SPLINE
SPL {X  -156.487, Y  +349.204, Z    +0.000, E1   -21.338, E3 -341381.497}
SPL {X  -159.136, Y  +365.992, Z    +0.000, E1   -12.463, E3 -341392.255}
SPL {X  -159.799, Y  +374.694, Z    +0.000, E1    -7.504, E3 -341395.359}
SPL {X  -159.976, Y  +380.404, Z    +0.000, E1    -3.959, E3 -341396.892}
SPL {X  -159.990, Y  +384.773, Z    +0.000, E1    -1.003, E3 -341397.786}
SPL {X  -159.990, Y  +387.968, Z    +0.000, E1    +1.448, E3 -341398.355}
SPL {X  -159.990, Y  +391.397, Z    +0.000, E1    +4.422, E3 -341398.979}
SPL {X  -159.990, Y  +395.864, Z    +0.000, E1    +8.712, E3 -341400.067}
SPL {X  -159.990, Y  +401.273, Z    +0.000, E1   +14.176, E3 -341401.795}
SPL {X  -159.990, Y  +411.788, Z    +0.000, E1   +23.693, E3 -341407.338}
SPL {X  -159.990, Y  +438.158, Z    +0.000, E1   +37.630, E3 -341430.615}
SPL {X  -159.990, Y  +468.567, Z    +0.000, E1   +41.922, E3 -341479.959}
SPL {X  -159.990, Y  +474.616, Z    +0.000, E1   +41.909, E3 -341494.288}
SPL {X  -159.990, Y  +481.610, Z    +0.000, E1   +41.947, E3 -341510.775}
SPL {X  -159.990, Y  +488.618, Z    +0.000, E1   +41.913, E3 -341527.387}
SPL {X  -159.990, Y  +494.299, Z    +0.000, E1   +41.910, E3 -341540.821}
SPL {X  -159.990, Y  +499.538, Z    +0.000, E1   +41.904, E3 -341553.216}
SPL {X  -159.990, Y  +505.259, Z    +0.000, E1   +41.922, E3 -341566.715}
SPL {X  -159.990, Y  +511.862, Z    +0.000, E1   +41.927, E3 -341582.325}
SPL {X  -159.990, Y  +517.450, Z    +0.000, E1   +41.901, E3 -341595.573}
SPL {X  -159.990, Y  +523.027, Z    +0.000, E1   +41.926, E3 -341608.717}
SPL {X  -159.990, Y  +528.611, Z    +0.000, E1   +41.900, E3 -341621.972}
SPL {X  -159.990, Y  +533.758, Z    +0.000, E1   +41.910, E3 -341634.121}
SPL {X  -159.990, Y  +539.474, Z    +0.000, E1   +41.912, E3 -341647.649}
SPL {X  -159.990, Y  +544.879, Z    +0.000, E1   +41.899, E3 -341660.460}
SPL {X  -159.990, Y  +550.802, Z    +0.000, E1   +41.920, E3 -341674.442}
SPL {X  -159.990, Y  +556.952, Z    +0.000, E1   +41.911, E3 -341688.981}
SPL {X  -159.990, Y  +562.629, Z    +0.000, E1   +41.910, E3 -341702.399}
SPL {X  -159.990, Y  +567.682, Z    +0.000, E1   +41.901, E3 -341714.358}
SPL {X  -159.990, Y  +572.912, Z    +0.000, E1   +41.914, E3 -341726.705}
SPL {X  -159.990, Y  +578.863, Z    +0.000, E1   +41.918, E3 -341740.769}
SPL {X  -159.990, Y  +584.320, Z    +0.000, E1   +41.901, E3 -341753.716}
SPL {X  -159.990, Y  +589.217, Z    +0.000, E1   +41.901, E3 -341765.289}
SPL {X  -159.990, Y  +594.252, Z    +0.000, E1   +41.903, E3 -341777.203}
SPL {X  -159.990, Y  +598.793, Z    +0.000, E1   +41.896, E3 -341787.957}
SPL {X  -159.990, Y  +604.215, Z    +0.000, E1   +41.919, E3 -341800.737}
SPL {X  -159.990, Y  +610.545, Z    +0.000, E1   +41.917, E3 -341815.707}
SPL {X  -159.990, Y  +615.720, Z    +0.000, E1   +41.899, E3 -341827.967}
SPL {X  -159.990, Y  +620.005, Z    +0.000, E1   +41.900, E3 -341838.100}
SPL {X  -159.990, Y  +624.919, Z    +0.000, E1   +41.912, E3 -341849.707}
SPL {X  -159.990, Y  +630.816, Z    +0.000, E1   +41.915, E3 -341863.636}
SPL {X  -159.990, Y  +637.009, Z    +0.000, E1   +41.925, E3 -341878.262}
SPL {X  -159.990, Y  +642.624, Z    +0.000, E1   +41.901, E3 -341891.583}
SPL {X  -159.990, Y  +647.782, Z    +0.000, E1   +41.914, E3 -341903.751}
SPL {X  -159.990, Y  +653.094, Z    +0.000, E1   +41.905, E3 -341916.329}
SPL {X  -159.990, Y  +657.893, Z    +0.000, E1   +41.899, E3 -341927.695}
SPL {X  -159.990, Y  +662.516, Z    +0.000, E1   +41.899, E3 -341938.626}
SPL {X  -159.990, Y  +668.411, Z    +0.000, E1   +41.929, E3 -341952.520}
SPL {X  -159.968, Y  +674.139, Z    +0.000, E1   +41.898, E3 -341966.124}
SPL {X  -159.817, Y  +678.937, Z    +0.000, E1   +41.879, E3 -341977.620}
SPL {X  -159.484, Y  +684.213, Z    +0.000, E1   +41.818, E3 -341990.456}
SPL {X  -159.007, Y  +689.209, Z    +0.000, E1   +41.732, E3 -342002.761}
SPL {X  -158.327, Y  +694.511, Z    +0.000, E1   +41.622, E3 -342016.012}
SPL {X  -157.480, Y  +699.729, Z    +0.000, E1   +41.453, E3 -342029.275}
SPL {X  -156.604, Y  +704.242, Z    +0.000, E1   +41.288, E3 -342040.884}
SPL {X  -155.514, Y  +709.078, Z    +0.000, E1   +41.107, E3 -342053.437}
SPL {X  -154.232, Y  +714.035, Z    +0.000, E1   +40.861, E3 -342066.496}
SPL {X  -153.147, Y  +717.790, Z    +0.000, E1   +40.640, E3 -342076.515}
SPL {X  -151.881, Y  +721.788, Z    +0.000, E1   +40.435, E3 -342087.201}
SPL {X  -148.572, Y  +730.857, Z    +0.000, E1   +36.304, E3 -342143.410}
ENDSPLINE

SPLINE
SPL {X  -156.377, Y  +705.307, Z    +0.000, E1   +21.740, E3 -342197.659}
SPL {X  -159.301, Y  +686.331, Z    +0.000, E1   +11.648, E3 -342210.303}
SPL {X  -159.936, Y  +675.651, Z    +0.000, E1    +5.377, E3 -342214.019}
SPL {X  -159.990, Y  +670.142, Z    +0.000, E1    +1.740, E3 -342215.318}
SPL {X  -159.990, Y  +666.629, Z    +0.000, E1    -0.827, E3 -342215.968}
SPL {X  -159.990, Y  +662.407, Z    +0.000, E1    -4.406, E3 -342216.818}
SPL {X  -159.990, Y  +657.382, Z    +0.000, E1    -9.217, E3 -342218.200}
SPL {X  -159.990, Y  +653.255, Z    +0.000, E1   -13.347, E3 -342219.529}
SPL {X  -159.990, Y  +646.242, Z    +0.000, E1   -19.956, E3 -342222.603}
SPL {X  -159.990, Y  +624.365, Z    +0.000, E1   -33.860, E3 -342240.504}
SPL {X  -159.990, Y  +615.596, Z    +0.000, E1   -36.980, E3 -342250.163}
SPL {X  -159.990, Y  +586.905, Z    +0.000, E1   -41.264, E3 -342297.189}
SPL {X  -159.990, Y  +581.111, Z    +0.000, E1   -41.245, E3 -342311.243}
SPL {X  -159.990, Y  +576.269, Z    +0.000, E1   -41.239, E3 -342322.971}
SPL {X  -159.990, Y  +571.714, Z    +0.000, E1   -41.240, E3 -342333.999}
SPL {X  -159.990, Y  +567.050, Z    +0.000, E1   -41.238, E3 -342345.286}
SPL {X  -159.990, Y  +561.959, Z    +0.000, E1   -41.251, E3 -342357.584}
SPL {X  -159.990, Y  +557.719, Z    +0.000, E1   -41.226, E3 -342367.886}
SPL {X  -159.990, Y  +554.148, Z    +0.000, E1   -41.237, E3 -342376.502}
SPL {X  -159.990, Y  +548.812, Z    +0.000, E1   -41.263, E3 -342389.376}
SPL {X  -159.990, Y  +543.804, Z    +0.000, E1   -41.237, E3 -342401.541}
SPL {X  -159.990, Y  +538.952, Z    +0.000, E1   -41.247, E3 -342413.288}
SPL {X  -159.990, Y  +534.225, Z    +0.000, E1   -41.236, E3 -342424.721}
SPL {X  -159.990, Y  +529.136, Z    +0.000, E1   -41.262, E3 -342436.997}
SPL {X  -159.990, Y  +522.690, Z    +0.000, E1   -41.265, E3 -342452.597}
SPL {X  -159.990, Y  +516.698, Z    +0.000, E1   -41.259, E3 -342467.071}
SPL {X  -159.990, Y  +510.896, Z    +0.000, E1   -41.267, E3 -342481.089}
SPL {X  -159.990, Y  +505.215, Z    +0.000, E1   -41.261, E3 -342494.849}
SPL {X  -159.990, Y  +500.102, Z    +0.000, E1   -41.251, E3 -342507.232}
SPL {X  -159.990, Y  +495.023, Z    +0.000, E1   -41.263, E3 -342519.481}
SPL {X  -159.990, Y  +479.011, Z    +0.000, E1   -45.740, E3 -342528.863}
SPL {X  -159.990, Y  +471.379, Z    +0.000, E1   -46.435, E3 -342540.479}
SPL {X  -159.990, Y  +465.881, Z    +0.000, E1   -45.385, E3 -342558.081}
SPL {X  -159.990, Y  +461.571, Z    +0.000, E1   -44.440, E3 -342572.607}
SPL {X  -159.990, Y  +458.229, Z    +0.000, E1   -43.579, E3 -342585.141}
SPL {X  -159.990, Y  +453.434, Z    +0.000, E1   -43.227, E3 -342597.915}
SPL {X  -159.990, Y  +448.702, Z    +0.000, E1   -43.218, E3 -342608.637}
SPL {X  -159.990, Y  +442.224, Z    +0.000, E1   -43.270, E3 -342623.187}
SPL {X  -159.990, Y  +435.724, Z    +0.000, E1   -43.218, E3 -342637.945}
SPL {X  -159.990, Y  +430.527, Z    +0.000, E1   -43.236, E3 -342649.634}
SPL {X  -159.990, Y  +424.433, Z    +0.000, E1   -43.237, E3 -342663.383}
SPL {X  -159.990, Y  +419.466, Z    +0.000, E1   -43.217, E3 -342674.623}
SPL {X  -159.990, Y  +414.585, Z    +0.000, E1   -43.233, E3 -342685.615}
SPL {X  -159.990, Y  +409.927, Z    +0.000, E1   -43.217, E3 -342696.147}
SPL {X  -159.990, Y  +405.428, Z    +0.000, E1   -43.230, E3 -342706.305}
SPL {X  -159.990, Y  +398.518, Z    +0.000, E1   -43.261, E3 -342721.859}
SPL {X  -159.990, Y  +392.163, Z    +0.000, E1   -43.223, E3 -342736.259}
SPL {X  -159.990, Y  +387.342, Z    +0.000, E1   -43.224, E3 -342747.137}
SPL {X  -159.990, Y  +382.548, Z    +0.000, E1   -43.224, E3 -342757.959}
SPL {X  -159.922, Y  +377.835, Z    +0.000, E1   -43.211, E3 -342768.676}
SPL {X  -159.712, Y  +373.072, Z    +0.000, E1   -43.177, E3 -342779.642}
SPL {X  -159.289, Y  +367.537, Z    +0.000, E1   -43.118, E3 -342792.554}
SPL {X  -158.730, Y  +362.464, Z    +0.000, E1   -43.003, E3 -342804.586}
SPL {X  -158.182, Y  +358.518, Z    +0.000, E1   -42.902, E3 -342814.064}
SPL {X  -157.507, Y  +354.423, Z    +0.000, E1   -42.786, E3 -342824.010}
SPL {X  -156.676, Y  +350.104, Z    +0.000, E1   -42.637, E3 -342834.615}
SPL {X  -155.489, Y  +344.819, Z    +0.000, E1   -42.446, E3 -342847.738}
SPL {X  -153.911, Y  +338.816, Z    +0.000, E1   -42.155, E3 -342862.914}
SPL {X  -152.412, Y  +333.846, Z    +0.000, E1   -41.856, E3 -342875.685}
SPL {X  -151.009, Y  +329.651, Z    +0.000, E1   -41.581, E3 -342886.585}
SPL {X  -148.356, Y  +322.607, Z    +0.000, E1   -36.121, E3 -342947.061}
ENDSPLINE

SPLINE
SPL {X  -156.487, Y  +349.204, Z    +0.000, E1   -21.338, E3 -343002.186}
SPL {X  -159.136, Y  +365.992, Z    +0.000, E1   -12.463, E3 -343012.945}
SPL {X  -159.799, Y  +374.694, Z    +0.000, E1    -7.504, E3 -343016.049}
SPL {X  -159.976, Y  +380.404, Z    +0.000, E1    -3.959, E3 -343017.582}
SPL {X  -159.990, Y  +384.773, Z    +0.000, E1    -1.003, E3 -343018.476}
SPL {X  -159.990, Y  +387.968, Z    +0.000, E1    +1.448, E3 -343019.044}
SPL {X  -159.990, Y  +391.397, Z    +0.000, E1    +4.422, E3 -343019.668}
SPL {X  -159.990, Y  +395.864, Z    +0.000, E1    +8.712, E3 -343020.757}
SPL {X  -159.990, Y  +401.273, Z    +0.000, E1   +14.176, E3 -343022.484}
SPL {X  -159.990, Y  +411.788, Z    +0.000, E1   +23.693, E3 -343028.027}
SPL {X  -159.990, Y  +438.158, Z    +0.000, E1   +37.630, E3 -343051.304}
SPL {X  -159.990, Y  +468.567, Z    +0.000, E1   +41.922, E3 -343100.648}
SPL {X  -159.990, Y  +474.616, Z    +0.000, E1   +41.909, E3 -343114.978}
SPL {X  -159.990, Y  +478.952, Z    +0.000, E1   +41.885, E3 -343125.276}
SPL {X  -159.990, Y  +484.724, Z    +0.000, E1   +41.943, E3 -343138.827}
SPL {X  -159.990, Y  +492.944, Z    +0.000, E1   +41.952, E3 -343158.247}
SPL {X  -159.990, Y  +499.538, Z    +0.000, E1   +41.904, E3 -343173.905}
SPL {X  -159.990, Y  +505.259, Z    +0.000, E1   +41.922, E3 -343187.405}
SPL {X  -159.990, Y  +511.862, Z    +0.000, E1   +41.927, E3 -343203.015}
SPL {X  -159.990, Y  +517.450, Z    +0.000, E1   +41.901, E3 -343216.262}
SPL {X  -159.990, Y  +523.027, Z    +0.000, E1   +41.926, E3 -343229.407}
SPL {X  -159.990, Y  +528.611, Z    +0.000, E1   +41.900, E3 -343242.662}
SPL {X  -159.990, Y  +533.758, Z    +0.000, E1   +41.910, E3 -343254.811}
SPL {X  -159.990, Y  +539.474, Z    +0.000, E1   +41.912, E3 -343268.338}
SPL {X  -159.990, Y  +544.879, Z    +0.000, E1   +41.899, E3 -343281.150}
SPL {X  -159.990, Y  +550.802, Z    +0.000, E1   +41.920, E3 -343295.131}
SPL {X  -159.990, Y  +556.952, Z    +0.000, E1   +41.911, E3 -343309.670}
SPL {X  -159.990, Y  +562.629, Z    +0.000, E1   +41.910, E3 -343323.088}
SPL {X  -159.990, Y  +569.054, Z    +0.000, E1   +41.933, E3 -343338.243}
SPL {X  -159.990, Y  +575.562, Z    +0.000, E1   +41.916, E3 -343353.656}
SPL {X  -159.990, Y  +580.118, Z    +0.000, E1   +41.891, E3 -343364.469}
SPL {X  -159.990, Y  +584.320, Z    +0.000, E1   +41.901, E3 -343374.405}
SPL {X  -159.990, Y  +589.217, Z    +0.000, E1   +41.901, E3 -343385.978}
SPL {X  -159.990, Y  +594.252, Z    +0.000, E1   +41.903, E3 -343397.893}
SPL {X  -159.990, Y  +598.793, Z    +0.000, E1   +41.896, E3 -343408.647}
SPL {X  -159.990, Y  +604.215, Z    +0.000, E1   +41.919, E3 -343421.427}
SPL {X  -159.990, Y  +609.216, Z    +0.000, E1   +41.890, E3 -343433.295}
SPL {X  -159.990, Y  +614.570, Z    +0.000, E1   +41.926, E3 -343445.900}
SPL {X  -159.990, Y  +620.005, Z    +0.000, E1   +41.900, E3 -343458.790}
SPL {X  -159.990, Y  +624.919, Z    +0.000, E1   +41.912, E3 -343470.397}
SPL {X  -159.990, Y  +630.816, Z    +0.000, E1   +41.915, E3 -343484.326}
SPL {X  -159.990, Y  +635.747, Z    +0.000, E1   +41.898, E3 -343496.005}
SPL {X  -159.990, Y  +641.479, Z    +0.000, E1   +41.931, E3 -343509.519}
SPL {X  -159.990, Y  +647.782, Z    +0.000, E1   +41.914, E3 -343524.441}
SPL {X  -159.990, Y  +653.094, Z    +0.000, E1   +41.905, E3 -343537.019}
SPL {X  -159.990, Y  +657.893, Z    +0.000, E1   +41.899, E3 -343548.385}
SPL {X  -159.990, Y  +662.516, Z    +0.000, E1   +41.899, E3 -343559.316}
SPL {X  -159.990, Y  +668.411, Z    +0.000, E1   +41.929, E3 -343573.210}
SPL {X  -159.968, Y  +674.139, Z    +0.000, E1   +41.898, E3 -343586.814}
SPL {X  -159.817, Y  +678.937, Z    +0.000, E1   +41.879, E3 -343598.310}
SPL {X  -159.484, Y  +684.213, Z    +0.000, E1   +41.818, E3 -343611.146}
SPL {X  -159.007, Y  +689.209, Z    +0.000, E1   +41.732, E3 -343623.451}
SPL {X  -158.327, Y  +694.511, Z    +0.000, E1   +41.622, E3 -343636.702}
SPL {X  -157.480, Y  +699.729, Z    +0.000, E1   +41.453, E3 -343649.965}
SPL {X  -156.604, Y  +704.242, Z    +0.000, E1   +41.288, E3 -343661.573}
SPL {X  -155.514, Y  +709.078, Z    +0.000, E1   +41.107, E3 -343674.127}
SPL {X  -154.232, Y  +714.035, Z    +0.000, E1   +40.861, E3 -343687.186}
SPL {X  -153.147, Y  +717.790, Z    +0.000, E1   +40.640, E3 -343697.204}
SPL {X  -151.881, Y  +721.788, Z    +0.000, E1   +40.435, E3 -343707.891}
SPL {X  -148.572, Y  +730.857, Z    +0.000, E1   +36.304, E3 -343764.100}
ENDSPLINE

SPLINE
SPL {X  -156.377, Y  +705.307, Z    +0.000, E1   +21.740, E3 -343818.348}
SPL {X  -158.965, Y  +689.585, Z    +0.000, E1   +13.405, E3 -343829.506}
SPL {X  -159.884, Y  +677.314, Z    +0.000, E1    +6.475, E3 -343834.219}
SPL {X  -159.990, Y  +670.142, Z    +0.000, E1    +1.740, E3 -343836.008}
SPL {X  -159.990, Y  +666.629, Z    +0.000, E1    -0.827, E3 -343836.658}
SPL {X  -159.990, Y  +662.407, Z    +0.000, E1    -4.406, E3 -343837.508}
SPL {X  -159.990, Y  +657.382, Z    +0.000, E1    -9.217, E3 -343838.890}
SPL {X  -159.990, Y  +653.255, Z    +0.000, E1   -13.347, E3 -343840.219}
SPL {X  -159.990, Y  +646.242, Z    +0.000, E1   -19.956, E3 -343843.293}
SPL {X  -159.990, Y  +624.365, Z    +0.000, E1   -33.860, E3 -343861.194}
SPL {X  -159.990, Y  +615.596, Z    +0.000, E1   -36.980, E3 -343870.853}
SPL {X  -159.990, Y  +586.905, Z    +0.000, E1   -41.264, E3 -343917.879}
SPL {X  -159.990, Y  +581.111, Z    +0.000, E1   -41.245, E3 -343931.933}
SPL {X  -159.990, Y  +576.269, Z    +0.000, E1   -41.239, E3 -343943.661}
SPL {X  -159.990, Y  +571.714, Z    +0.000, E1   -41.240, E3 -343954.689}
SPL {X  -159.990, Y  +567.050, Z    +0.000, E1   -41.238, E3 -343965.975}
SPL {X  -159.990, Y  +561.959, Z    +0.000, E1   -41.251, E3 -343978.274}
SPL {X  -159.990, Y  +555.553, Z    +0.000, E1   -41.273, E3 -343993.742}
SPL {X  -159.990, Y  +549.897, Z    +0.000, E1   -41.240, E3 -344007.472}
SPL {X  -159.990, Y  +544.775, Z    +0.000, E1   -41.260, E3 -344019.847}
SPL {X  -159.990, Y  +540.176, Z    +0.000, E1   -41.224, E3 -344031.056}
SPL {X  -159.990, Y  +535.325, Z    +0.000, E1   -41.260, E3 -344042.719}
SPL {X  -159.990, Y  +529.136, Z    +0.000, E1   -41.262, E3 -344057.687}
SPL {X  -159.990, Y  +522.690, Z    +0.000, E1   -41.265, E3 -344073.287}
SPL {X  -159.990, Y  +516.698, Z    +0.000, E1   -41.259, E3 -344087.761}
SPL {X  -159.990, Y  +510.896, Z    +0.000, E1   -41.267, E3 -344101.779}
SPL {X  -159.990, Y  +505.215, Z    +0.000, E1   -41.261, E3 -344115.539}
SPL {X  -159.990, Y  +500.102, Z    +0.000, E1   -41.251, E3 -344127.922}
SPL {X  -159.990, Y  +495.023, Z    +0.000, E1   -41.263, E3 -344140.171}
SPL {X  -159.990, Y  +479.011, Z    +0.000, E1   -45.740, E3 -344149.553}
SPL {X  -159.990, Y  +471.379, Z    +0.000, E1   -46.435, E3 -344161.168}
SPL {X  -159.990, Y  +466.895, Z    +0.000, E1   -45.533, E3 -344175.573}
SPL {X  -159.990, Y  +462.409, Z    +0.000, E1   -44.664, E3 -344190.348}
SPL {X  -159.990, Y  +458.229, Z    +0.000, E1   -43.579, E3 -344205.830}
SPL {X  -159.990, Y  +453.434, Z    +0.000, E1   -43.227, E3 -344218.605}
SPL {X  -159.990, Y  +448.702, Z    +0.000, E1   -43.218, E3 -344229.326}
SPL {X  -159.990, Y  +442.224, Z    +0.000, E1   -43.270, E3 -344243.876}
SPL {X  -159.990, Y  +435.724, Z    +0.000, E1   -43.218, E3 -344258.634}
SPL {X  -159.990, Y  +430.527, Z    +0.000, E1   -43.236, E3 -344270.324}
SPL {X  -159.990, Y  +424.433, Z    +0.000, E1   -43.237, E3 -344284.073}
SPL {X  -159.990, Y  +419.466, Z    +0.000, E1   -43.217, E3 -344295.313}
SPL {X  -159.990, Y  +414.585, Z    +0.000, E1   -43.233, E3 -344306.305}
SPL {X  -159.990, Y  +409.927, Z    +0.000, E1   -43.217, E3 -344316.836}
SPL {X  -159.990, Y  +405.428, Z    +0.000, E1   -43.230, E3 -344326.994}
SPL {X  -159.990, Y  +398.518, Z    +0.000, E1   -43.261, E3 -344342.549}
SPL {X  -159.990, Y  +392.163, Z    +0.000, E1   -43.223, E3 -344356.949}
SPL {X  -159.990, Y  +387.342, Z    +0.000, E1   -43.224, E3 -344367.826}
SPL {X  -159.990, Y  +382.548, Z    +0.000, E1   -43.224, E3 -344378.649}
SPL {X  -159.922, Y  +377.835, Z    +0.000, E1   -43.211, E3 -344389.366}
SPL {X  -159.712, Y  +373.072, Z    +0.000, E1   -43.177, E3 -344400.332}
SPL {X  -159.289, Y  +367.537, Z    +0.000, E1   -43.118, E3 -344413.243}
SPL {X  -158.730, Y  +362.464, Z    +0.000, E1   -43.003, E3 -344425.275}
SPL {X  -158.182, Y  +358.518, Z    +0.000, E1   -42.902, E3 -344434.754}
SPL {X  -157.507, Y  +354.423, Z    +0.000, E1   -42.786, E3 -344444.699}
SPL {X  -156.676, Y  +350.104, Z    +0.000, E1   -42.637, E3 -344455.305}
SPL {X  -155.489, Y  +344.819, Z    +0.000, E1   -42.446, E3 -344468.428}
SPL {X  -153.911, Y  +338.816, Z    +0.000, E1   -42.155, E3 -344483.604}
SPL {X  -152.412, Y  +333.846, Z    +0.000, E1   -41.856, E3 -344496.375}
SPL {X  -151.009, Y  +329.651, Z    +0.000, E1   -41.581, E3 -344507.275}
SPL {X  -148.356, Y  +322.607, Z    +0.000, E1   -36.121, E3 -344567.750}
ENDSPLINE

SPLINE
SPL {X  -156.487, Y  +349.204, Z    +0.000, E1   -21.338, E3 -344622.876}
SPL {X  -159.136, Y  +365.992, Z    +0.000, E1   -12.463, E3 -344633.635}
SPL {X  -159.799, Y  +374.694, Z    +0.000, E1    -7.504, E3 -344636.738}
SPL {X  -159.976, Y  +380.404, Z    +0.000, E1    -3.959, E3 -344638.271}
SPL {X  -159.990, Y  +384.773, Z    +0.000, E1    -1.003, E3 -344639.166}
SPL {X  -159.990, Y  +387.968, Z    +0.000, E1    +1.448, E3 -344639.734}
SPL {X  -159.990, Y  +391.397, Z    +0.000, E1    +4.422, E3 -344640.358}
SPL {X  -159.990, Y  +395.864, Z    +0.000, E1    +8.712, E3 -344641.446}
SPL {X  -159.990, Y  +401.273, Z    +0.000, E1   +14.176, E3 -344643.174}
SPL {X  -159.990, Y  +409.369, Z    +0.000, E1   +21.807, E3 -344646.966}
SPL {X  -159.990, Y  +436.107, Z    +0.000, E1   +36.921, E3 -344669.891}
SPL {X  -159.990, Y  +465.724, Z    +0.000, E1   +41.883, E3 -344714.689}
SPL {X  -159.990, Y  +470.837, Z    +0.000, E1   +41.927, E3 -344726.703}
SPL {X  -159.990, Y  +477.498, Z    +0.000, E1   +41.916, E3 -344742.479}
SPL {X  -159.990, Y  +483.140, Z    +0.000, E1   +41.902, E3 -344755.835}
SPL {X  -159.990, Y  +488.618, Z    +0.000, E1   +41.913, E3 -344768.766}
SPL {X  -159.990, Y  +494.299, Z    +0.000, E1   +41.910, E3 -344782.201}
SPL {X  -159.990, Y  +499.538, Z    +0.000, E1   +41.904, E3 -344794.595}
SPL {X  -159.990, Y  +505.259, Z    +0.000, E1   +41.922, E3 -344808.094}
SPL {X  -159.990, Y  +511.862, Z    +0.000, E1   +41.927, E3 -344823.704}
SPL {X  -159.990, Y  +517.450, Z    +0.000, E1   +41.901, E3 -344836.952}
SPL {X  -159.990, Y  +523.027, Z    +0.000, E1   +41.926, E3 -344850.096}
SPL {X  -159.990, Y  +528.611, Z    +0.000, E1   +41.900, E3 -344863.351}
SPL {X  -159.990, Y  +533.758, Z    +0.000, E1   +41.910, E3 -344875.501}
SPL {X  -159.990, Y  +539.474, Z    +0.000, E1   +41.912, E3 -344889.028}
SPL {X  -159.990, Y  +544.879, Z    +0.000, E1   +41.899, E3 -344901.840}
SPL {X  -159.990, Y  +550.802, Z    +0.000, E1   +41.920, E3 -344915.821}
SPL {X  -159.990, Y  +556.952, Z    +0.000, E1   +41.911, E3 -344930.360}
SPL {X  -159.990, Y  +562.629, Z    +0.000, E1   +41.910, E3 -344943.778}
SPL {X  -159.990, Y  +567.682, Z    +0.000, E1   +41.901, E3 -344955.737}
SPL {X  -159.990, Y  +572.912, Z    +0.000, E1   +41.914, E3 -344968.084}
SPL {X  -159.990, Y  +578.863, Z    +0.000, E1   +41.918, E3 -344982.148}
SPL {X  -159.990, Y  +584.320, Z    +0.000, E1   +41.901, E3 -344995.095}
SPL {X  -159.990, Y  +589.217, Z    +0.000, E1   +41.901, E3 -345006.668}
SPL {X  -159.990, Y  +594.252, Z    +0.000, E1   +41.903, E3 -345018.582}
SPL {X  -159.990, Y  +598.793, Z    +0.000, E1   +41.896, E3 -345029.336}
SPL {X  -159.990, Y  +604.215, Z    +0.000, E1   +41.919, E3 -345042.117}
SPL {X  -159.990, Y  +609.216, Z    +0.000, E1   +41.890, E3 -345053.985}
SPL {X  -159.990, Y  +614.570, Z    +0.000, E1   +41.926, E3 -345066.590}
SPL {X  -159.990, Y  +620.005, Z    +0.000, E1   +41.900, E3 -345079.479}
SPL {X  -159.990, Y  +624.919, Z    +0.000, E1   +41.912, E3 -345091.087}
SPL {X  -159.990, Y  +629.282, Z    +0.000, E1   +41.888, E3 -345101.427}
SPL {X  -159.990, Y  +632.270, Z    +0.000, E1   +41.887, E3 -345108.499}
SPL {X  -159.990, Y  +637.009, Z    +0.000, E1   +41.925, E3 -345119.641}
SPL {X  -159.990, Y  +642.624, Z    +0.000, E1   +41.901, E3 -345132.962}
SPL {X  -159.990, Y  +647.782, Z    +0.000, E1   +41.914, E3 -345145.130}
SPL {X  -159.990, Y  +653.094, Z    +0.000, E1   +41.905, E3 -345157.709}
SPL {X  -159.990, Y  +657.893, Z    +0.000, E1   +41.899, E3 -345169.074}
SPL {X  -159.990, Y  +662.516, Z    +0.000, E1   +41.899, E3 -345180.006}
SPL {X  -159.990, Y  +668.411, Z    +0.000, E1   +41.929, E3 -345193.899}
SPL {X  -159.968, Y  +674.139, Z    +0.000, E1   +41.898, E3 -345207.503}
SPL {X  -159.817, Y  +678.937, Z    +0.000, E1   +41.879, E3 -345218.999}
SPL {X  -159.484, Y  +684.213, Z    +0.000, E1   +41.818, E3 -345231.836}
SPL {X  -159.007, Y  +689.209, Z    +0.000, E1   +41.732, E3 -345244.141}
SPL {X  -158.327, Y  +694.511, Z    +0.000, E1   +41.622, E3 -345257.391}
SPL {X  -157.480, Y  +699.729, Z    +0.000, E1   +41.453, E3 -345270.654}
SPL {X  -156.604, Y  +704.242, Z    +0.000, E1   +41.288, E3 -345282.263}
SPL {X  -155.831, Y  +707.744, Z    +0.000, E1   +41.132, E3 -345291.383}
SPL {X  -155.167, Y  +710.488, Z    +0.000, E1   +41.008, E3 -345298.561}
SPL {X  -154.232, Y  +714.035, Z    +0.000, E1   +40.861, E3 -345307.876}
SPL {X  -153.147, Y  +717.790, Z    +0.000, E1   +40.640, E3 -345317.894}
SPL {X  -151.881, Y  +721.788, Z    +0.000, E1   +40.435, E3 -345328.580}
SPL {X  -148.572, Y  +730.857, Z    +0.000, E1   +36.304, E3 -345384.789}
ENDSPLINE

SPLINE
SPL {X  -156.377, Y  +705.307, Z    +0.000, E1   +21.740, E3 -345439.038}
SPL {X  -158.965, Y  +689.585, Z    +0.000, E1   +13.405, E3 -345450.196}
SPL {X  -159.884, Y  +677.314, Z    +0.000, E1    +6.475, E3 -345454.908}
SPL {X  -159.990, Y  +670.142, Z    +0.000, E1    +1.740, E3 -345456.698}
SPL {X  -159.990, Y  +666.629, Z    +0.000, E1    -0.827, E3 -345457.347}
SPL {X  -159.990, Y  +662.407, Z    +0.000, E1    -4.406, E3 -345458.198}
SPL {X  -159.990, Y  +657.382, Z    +0.000, E1    -9.217, E3 -345459.580}
SPL {X  -159.990, Y  +653.255, Z    +0.000, E1   -13.347, E3 -345460.909}
SPL {X  -159.990, Y  +646.242, Z    +0.000, E1   -19.956, E3 -345463.982}
SPL {X  -159.990, Y  +624.365, Z    +0.000, E1   -33.860, E3 -345481.884}
SPL {X  -159.990, Y  +615.596, Z    +0.000, E1   -36.980, E3 -345491.542}
SPL {X  -159.990, Y  +588.349, Z    +0.000, E1   -41.235, E3 -345535.121}
SPL {X  -159.990, Y  +582.302, Z    +0.000, E1   -41.281, E3 -345549.688}
SPL {X  -159.990, Y  +576.269, Z    +0.000, E1   -41.239, E3 -345564.350}
SPL {X  -159.990, Y  +571.714, Z    +0.000, E1   -41.240, E3 -345575.378}
SPL {X  -159.990, Y  +567.050, Z    +0.000, E1   -41.238, E3 -345586.665}
SPL {X  -159.990, Y  +561.959, Z    +0.000, E1   -41.251, E3 -345598.963}
SPL {X  -159.990, Y  +555.553, Z    +0.000, E1   -41.273, E3 -345614.432}
SPL {X  -159.990, Y  +549.897, Z    +0.000, E1   -41.240, E3 -345628.162}
SPL {X  -159.990, Y  +544.775, Z    +0.000, E1   -41.260, E3 -345640.537}
SPL {X  -159.990, Y  +538.952, Z    +0.000, E1   -41.247, E3 -345654.668}
SPL {X  -159.990, Y  +532.945, Z    +0.000, E1   -41.264, E3 -345669.156}
SPL {X  -159.990, Y  +526.579, Z    +0.000, E1   -41.262, E3 -345684.568}
SPL {X  -159.990, Y  +521.454, Z    +0.000, E1   -41.236, E3 -345697.012}
SPL {X  -159.990, Y  +516.698, Z    +0.000, E1   -41.259, E3 -345708.451}
SPL {X  -159.990, Y  +510.896, Z    +0.000, E1   -41.267, E3 -345722.468}
SPL {X  -159.990, Y  +505.215, Z    +0.000, E1   -41.261, E3 -345736.228}
SPL {X  -159.990, Y  +498.837, Z    +0.000, E1   -41.283, E3 -345751.617}
SPL {X  -159.990, Y  +493.848, Z    +0.000, E1   -41.241, E3 -345763.737}
SPL {X  -159.990, Y  +474.734, Z    +0.000, E1   -46.319, E3 -345775.660}
SPL {X  -159.990, Y  +469.870, Z    +0.000, E1   -46.059, E3 -345786.883}
SPL {X  -159.990, Y  +465.881, Z    +0.000, E1   -45.385, E3 -345799.461}
SPL {X  -159.990, Y  +461.571, Z    +0.000, E1   -44.440, E3 -345813.986}
SPL {X  -159.990, Y  +458.229, Z    +0.000, E1   -43.579, E3 -345826.520}
SPL {X  -159.990, Y  +453.434, Z    +0.000, E1   -43.227, E3 -345839.294}
SPL {X  -159.990, Y  +448.702, Z    +0.000, E1   -43.218, E3 -345850.016}
SPL {X  -159.990, Y  +442.224, Z    +0.000, E1   -43.270, E3 -345864.566}
SPL {X  -159.990, Y  +435.724, Z    +0.000, E1   -43.218, E3 -345879.324}
SPL {X  -159.990, Y  +430.527, Z    +0.000, E1   -43.236, E3 -345891.014}
SPL {X  -159.990, Y  +424.433, Z    +0.000, E1   -43.237, E3 -345904.763}
SPL {X  -159.990, Y  +419.466, Z    +0.000, E1   -43.217, E3 -345916.002}
SPL {X  -159.990, Y  +414.585, Z    +0.000, E1   -43.233, E3 -345926.994}
SPL {X  -159.990, Y  +409.927, Z    +0.000, E1   -43.217, E3 -345937.526}
SPL {X  -159.990, Y  +405.428, Z    +0.000, E1   -43.230, E3 -345947.684}
SPL {X  -159.990, Y  +398.518, Z    +0.000, E1   -43.261, E3 -345963.238}
SPL {X  -159.990, Y  +392.163, Z    +0.000, E1   -43.223, E3 -345977.638}
SPL {X  -159.990, Y  +387.342, Z    +0.000, E1   -43.224, E3 -345988.516}
SPL {X  -159.990, Y  +382.548, Z    +0.000, E1   -43.224, E3 -345999.339}
SPL {X  -159.922, Y  +377.835, Z    +0.000, E1   -43.211, E3 -346010.055}
SPL {X  -159.712, Y  +373.072, Z    +0.000, E1   -43.177, E3 -346021.021}
SPL {X  -159.289, Y  +367.537, Z    +0.000, E1   -43.118, E3 -346033.933}
SPL {X  -158.730, Y  +362.464, Z    +0.000, E1   -43.003, E3 -346045.965}
SPL {X  -158.182, Y  +358.518, Z    +0.000, E1   -42.902, E3 -346055.444}
SPL {X  -157.507, Y  +354.423, Z    +0.000, E1   -42.786, E3 -346065.389}
SPL {X  -156.676, Y  +350.104, Z    +0.000, E1   -42.637, E3 -346075.994}
SPL {X  -155.807, Y  +346.154, Z    +0.000, E1   -42.470, E3 -346085.821}
SPL {X  -154.777, Y  +341.993, Z    +0.000, E1   -42.302, E3 -346096.246}
SPL {X  -153.585, Y  +337.686, Z    +0.000, E1   -42.062, E3 -346107.222}
SPL {X  -152.412, Y  +333.846, Z    +0.000, E1   -41.856, E3 -346117.064}
SPL {X  -151.009, Y  +329.651, Z    +0.000, E1   -41.581, E3 -346127.964}
SPL {X  -148.356, Y  +322.607, Z    +0.000, E1   -36.121, E3 -346188.440}
ENDSPLINE

SPLINE
SPL {X  -156.487, Y  +349.204, Z    +0.000, E1   -21.338, E3 -346243.566}
SPL {X  -159.136, Y  +365.992, Z    +0.000, E1   -12.463, E3 -346254.324}
SPL {X  -159.799, Y  +374.694, Z    +0.000, E1    -7.504, E3 -346257.428}
SPL {X  -159.976, Y  +380.404, Z    +0.000, E1    -3.959, E3 -346258.961}
SPL {X  -159.990, Y  +384.773, Z    +0.000, E1    -1.003, E3 -346259.855}
SPL {X  -159.990, Y  +387.968, Z    +0.000, E1    +1.448, E3 -346260.424}
SPL {X  -159.990, Y  +391.397, Z    +0.000, E1    +4.422, E3 -346261.048}
SPL {X  -159.990, Y  +395.864, Z    +0.000, E1    +8.712, E3 -346262.136}
SPL {X  -159.990, Y  +401.273, Z    +0.000, E1   +14.176, E3 -346263.864}
SPL {X  -159.990, Y  +409.369, Z    +0.000, E1   +21.807, E3 -346267.655}
SPL {X  -159.990, Y  +436.107, Z    +0.000, E1   +36.921, E3 -346290.581}
SPL {X  -159.990, Y  +468.567, Z    +0.000, E1   +41.922, E3 -346342.028}
SPL {X  -159.990, Y  +474.616, Z    +0.000, E1   +41.909, E3 -346356.357}
SPL {X  -159.990, Y  +478.952, Z    +0.000, E1   +41.885, E3 -346366.655}
SPL {X  -159.990, Y  +484.724, Z    +0.000, E1   +41.943, E3 -346380.207}
SPL {X  -159.990, Y  +492.944, Z    +0.000, E1   +41.952, E3 -346399.626}
SPL {X  -159.990, Y  +499.538, Z    +0.000, E1   +41.904, E3 -346415.285}
SPL {X  -159.990, Y  +505.259, Z    +0.000, E1   +41.922, E3 -346428.784}
SPL {X  -159.990, Y  +511.862, Z    +0.000, E1   +41.927, E3 -346444.394}
SPL {X  -159.990, Y  +519.146, Z    +0.000, E1   +41.942, E3 -346461.588}
SPL {X  -159.990, Y  +526.974, Z    +0.000, E1   +41.950, E3 -346480.088}
SPL {X  -159.990, Y  +533.758, Z    +0.000, E1   +41.910, E3 -346496.190}
SPL {X  -159.990, Y  +539.474, Z    +0.000, E1   +41.912, E3 -346509.718}
SPL {X  -159.990, Y  +546.447, Z    +0.000, E1   +41.939, E3 -346526.181}
SPL {X  -159.990, Y  +552.220, Z    +0.000, E1   +41.887, E3 -346539.914}
SPL {X  -159.990, Y  +556.952, Z    +0.000, E1   +41.911, E3 -346551.050}
SPL {X  -159.990, Y  +562.629, Z    +0.000, E1   +41.910, E3 -346564.468}
SPL {X  -159.990, Y  +567.682, Z    +0.000, E1   +41.901, E3 -346576.427}
SPL {X  -159.990, Y  +572.912, Z    +0.000, E1   +41.914, E3 -346588.774}
SPL {X  -159.990, Y  +578.863, Z    +0.000, E1   +41.918, E3 -346602.838}
SPL {X  -159.990, Y  +584.320, Z    +0.000, E1   +41.901, E3 -346615.785}
SPL {X  -159.990, Y  +589.217, Z    +0.000, E1   +41.901, E3 -346627.358}
SPL {X  -159.990, Y  +594.252, Z    +0.000, E1   +41.903, E3 -346639.272}
SPL {X  -159.990, Y  +598.793, Z    +0.000, E1   +41.896, E3 -346650.026}
SPL {X  -159.990, Y  +604.215, Z    +0.000, E1   +41.919, E3 -346662.806}
SPL {X  -159.990, Y  +610.545, Z    +0.000, E1   +41.917, E3 -346677.776}
SPL {X  -159.990, Y  +615.720, Z    +0.000, E1   +41.899, E3 -346690.036}
SPL {X  -159.990, Y  +621.417, Z    +0.000, E1   +41.931, E3 -346703.473}
SPL {X  -159.990, Y  +627.900, Z    +0.000, E1   +41.914, E3 -346718.812}
SPL {X  -159.990, Y  +634.411, Z    +0.000, E1   +41.931, E3 -346734.182}
SPL {X  -159.990, Y  +641.479, Z    +0.000, E1   +41.931, E3 -346750.898}
SPL {X  -159.990, Y  +647.782, Z    +0.000, E1   +41.914, E3 -346765.820}
SPL {X  -159.990, Y  +653.094, Z    +0.000, E1   +41.905, E3 -346778.398}
SPL {X  -159.990, Y  +657.893, Z    +0.000, E1   +41.899, E3 -346789.764}
SPL {X  -159.990, Y  +662.516, Z    +0.000, E1   +41.899, E3 -346800.695}
SPL {X  -159.990, Y  +668.411, Z    +0.000, E1   +41.929, E3 -346814.589}
SPL {X  -159.968, Y  +674.139, Z    +0.000, E1   +41.898, E3 -346828.193}
SPL {X  -159.817, Y  +678.937, Z    +0.000, E1   +41.879, E3 -346839.689}
SPL {X  -159.484, Y  +684.213, Z    +0.000, E1   +41.818, E3 -346852.525}
SPL {X  -159.007, Y  +689.209, Z    +0.000, E1   +41.732, E3 -346864.830}
SPL {X  -158.327, Y  +694.511, Z    +0.000, E1   +41.622, E3 -346878.081}
SPL {X  -157.480, Y  +699.729, Z    +0.000, E1   +41.453, E3 -346891.344}
SPL {X  -156.604, Y  +704.242, Z    +0.000, E1   +41.288, E3 -346902.953}
SPL {X  -155.514, Y  +709.078, Z    +0.000, E1   +41.107, E3 -346915.506}
SPL {X  -154.232, Y  +714.035, Z    +0.000, E1   +40.861, E3 -346928.565}
SPL {X  -153.147, Y  +717.790, Z    +0.000, E1   +40.640, E3 -346938.584}
SPL {X  -151.881, Y  +721.788, Z    +0.000, E1   +40.435, E3 -346949.270}
SPL {X  -148.572, Y  +730.857, Z    +0.000, E1   +36.304, E3 -347005.479}
ENDSPLINE

SPLINE
SPL {X  -154.420, Y  +713.347, Z    +0.000, E1   +25.698, E3 -347050.903}
SPL {X  -156.970, Y  +702.437, Z    +0.000, E1   +20.224, E3 -347062.599}
SPL {X  -159.301, Y  +686.331, Z    +0.000, E1   +11.648, E3 -347072.372}
SPL {X  -159.936, Y  +675.651, Z    +0.000, E1    +5.377, E3 -347076.088}
SPL {X  -159.990, Y  +670.142, Z    +0.000, E1    +1.740, E3 -347077.387}
SPL {X  -159.990, Y  +666.629, Z    +0.000, E1    -0.827, E3 -347078.037}
SPL {X  -159.990, Y  +662.407, Z    +0.000, E1    -4.406, E3 -347078.887}
SPL {X  -159.990, Y  +655.884, Z    +0.000, E1   -10.601, E3 -347080.753}
SPL {X  -159.990, Y  +643.833, Z    +0.000, E1   -21.883, E3 -347086.382}
SPL {X  -159.990, Y  +617.235, Z    +0.000, E1   -36.481, E3 -347110.282}
SPL {X  -159.990, Y  +586.905, Z    +0.000, E1   -41.264, E3 -347159.258}
SPL {X  -159.990, Y  +581.111, Z    +0.000, E1   -41.245, E3 -347173.312}
SPL {X  -159.990, Y  +576.269, Z    +0.000, E1   -41.239, E3 -347185.040}
SPL {X  -159.990, Y  +571.714, Z    +0.000, E1   -41.240, E3 -347196.068}
SPL {X  -159.990, Y  +567.050, Z    +0.000, E1   -41.238, E3 -347207.355}
SPL {X  -159.990, Y  +561.959, Z    +0.000, E1   -41.251, E3 -347219.653}
SPL {X  -159.990, Y  +555.553, Z    +0.000, E1   -41.273, E3 -347235.121}
SPL {X  -159.990, Y  +549.897, Z    +0.000, E1   -41.240, E3 -347248.852}
SPL {X  -159.990, Y  +544.775, Z    +0.000, E1   -41.260, E3 -347261.226}
SPL {X  -159.990, Y  +538.952, Z    +0.000, E1   -41.247, E3 -347275.357}
SPL {X  -159.990, Y  +534.225, Z    +0.000, E1   -41.236, E3 -347286.790}
SPL {X  -159.990, Y  +529.136, Z    +0.000, E1   -41.262, E3 -347299.066}
SPL {X  -159.990, Y  +524.776, Z    +0.000, E1   -41.225, E3 -347309.680}
SPL {X  -159.990, Y  +521.454, Z    +0.000, E1   -41.236, E3 -347317.702}
SPL {X  -159.990, Y  +515.605, Z    +0.000, E1   -41.288, E3 -347331.741}
SPL {X  -159.990, Y  +509.898, Z    +0.000, E1   -41.246, E3 -347345.602}
SPL {X  -159.990, Y  +505.215, Z    +0.000, E1   -41.261, E3 -347356.918}
SPL {X  -159.990, Y  +500.102, Z    +0.000, E1   -41.251, E3 -347369.301}
SPL {X  -159.990, Y  +495.023, Z    +0.000, E1   -41.263, E3 -347381.550}
SPL {X  -159.990, Y  +479.011, Z    +0.000, E1   -45.740, E3 -347390.932}
SPL {X  -159.990, Y  +471.379, Z    +0.000, E1   -46.435, E3 -347402.548}
SPL {X  -159.990, Y  +466.895, Z    +0.000, E1   -45.533, E3 -347416.952}
SPL {X  -159.990, Y  +462.409, Z    +0.000, E1   -44.664, E3 -347431.727}
SPL {X  -159.990, Y  +458.229, Z    +0.000, E1   -43.579, E3 -347447.210}
SPL {X  -159.990, Y  +453.434, Z    +0.000, E1   -43.227, E3 -347459.984}
SPL {X  -159.990, Y  +448.702, Z    +0.000, E1   -43.218, E3 -347470.706}
SPL {X  -159.990, Y  +444.476, Z    +0.000, E1   -43.219, E3 -347480.244}
SPL {X  -159.990, Y  +440.246, Z    +0.000, E1   -43.217, E3 -347489.802}
SPL {X  -159.990, Y  +434.411, Z    +0.000, E1   -43.246, E3 -347502.932}
SPL {X  -159.990, Y  +429.216, Z    +0.000, E1   -43.210, E3 -347514.704}
SPL {X  -159.990, Y  +424.433, Z    +0.000, E1   -43.237, E3 -347525.452}
SPL {X  -159.990, Y  +419.466, Z    +0.000, E1   -43.217, E3 -347536.692}
SPL {X  -159.990, Y  +414.585, Z    +0.000, E1   -43.233, E3 -347547.684}
SPL {X  -159.990, Y  +409.927, Z    +0.000, E1   -43.217, E3 -347558.215}
SPL {X  -159.990, Y  +405.428, Z    +0.000, E1   -43.230, E3 -347568.374}
SPL {X  -159.990, Y  +401.033, Z    +0.000, E1   -43.209, E3 -347578.328}
SPL {X  -159.990, Y  +396.968, Z    +0.000, E1   -43.221, E3 -347587.486}
SPL {X  -159.990, Y  +392.163, Z    +0.000, E1   -43.223, E3 -347598.328}
SPL {X  -159.990, Y  +387.342, Z    +0.000, E1   -43.224, E3 -347609.206}
SPL {X  -159.990, Y  +382.548, Z    +0.000, E1   -43.224, E3 -347620.028}
SPL {X  -159.922, Y  +377.835, Z    +0.000, E1   -43.211, E3 -347630.745}
SPL {X  -159.712, Y  +373.072, Z    +0.000, E1   -43.177, E3 -347641.711}
SPL {X  -159.289, Y  +367.537, Z    +0.000, E1   -43.118, E3 -347654.623}
SPL {X  -158.730, Y  +362.464, Z    +0.000, E1   -43.003, E3 -347666.655}
SPL {X  -158.182, Y  +358.518, Z    +0.000, E1   -42.902, E3 -347676.133}
SPL {X  -157.507, Y  +354.423, Z    +0.000, E1   -42.786, E3 -347686.079}
SPL {X  -156.676, Y  +350.104, Z    +0.000, E1   -42.637, E3 -347696.684}
SPL {X  -155.807, Y  +346.154, Z    +0.000, E1   -42.470, E3 -347706.511}
SPL {X  -154.777, Y  +341.993, Z    +0.000, E1   -42.302, E3 -347716.936}
SPL {X  -153.585, Y  +337.686, Z    +0.000, E1   -42.062, E3 -347727.911}
SPL {X  -152.412, Y  +333.846, Z    +0.000, E1   -41.856, E3 -347737.754}
SPL {X  -151.009, Y  +329.651, Z    +0.000, E1   -41.581, E3 -347748.654}
SPL {X  -148.356, Y  +322.607, Z    +0.000, E1   -36.121, E3 -347809.129}
ENDSPLINE

SPLINE
SPL {X  -156.487, Y  +349.204, Z    +0.000, E1   -21.338, E3 -347864.255}
SPL {X  -159.136, Y  +365.992, Z    +0.000, E1   -12.463, E3 -347875.014}
SPL {X  -159.799, Y  +374.694, Z    +0.000, E1    -7.504, E3 -347878.118}
SPL {X  -159.976, Y  +380.404, Z    +0.000, E1    -3.959, E3 -347879.651}
SPL {X  -159.990, Y  +384.773, Z    +0.000, E1    -1.003, E3 -347880.545}
SPL {X  -159.990, Y  +387.968, Z    +0.000, E1    +1.448, E3 -347881.113}
SPL {X  -159.990, Y  +391.397, Z    +0.000, E1    +4.422, E3 -347881.737}
SPL {X  -159.990, Y  +395.864, Z    +0.000, E1    +8.712, E3 -347882.826}
SPL {X  -159.990, Y  +401.273, Z    +0.000, E1   +14.176, E3 -347884.553}
SPL {X  -159.990, Y  +409.369, Z    +0.000, E1   +21.807, E3 -347888.345}
SPL {X  -159.990, Y  +436.107, Z    +0.000, E1   +36.921, E3 -347911.270}
SPL {X  -159.990, Y  +465.724, Z    +0.000, E1   +41.883, E3 -347956.068}
SPL {X  -159.990, Y  +470.837, Z    +0.000, E1   +41.927, E3 -347968.083}
SPL {X  -159.990, Y  +477.498, Z    +0.000, E1   +41.916, E3 -347983.858}
SPL {X  -159.990, Y  +484.724, Z    +0.000, E1   +41.943, E3 -348000.896}
SPL {X  -159.990, Y  +492.944, Z    +0.000, E1   +41.952, E3 -348020.316}
SPL {X  -159.990, Y  +499.538, Z    +0.000, E1   +41.904, E3 -348035.974}
SPL {X  -159.990, Y  +505.259, Z    +0.000, E1   +41.922, E3 -348049.474}
SPL {X  -159.990, Y  +511.862, Z    +0.000, E1   +41.927, E3 -348065.084}
SPL {X  -159.990, Y  +517.450, Z    +0.000, E1   +41.901, E3 -348078.331}
SPL {X  -159.990, Y  +523.027, Z    +0.000, E1   +41.926, E3 -348091.476}
SPL {X  -159.990, Y  +528.611, Z    +0.000, E1   +41.900, E3 -348104.731}
SPL {X  -159.990, Y  +533.758, Z    +0.000, E1   +41.910, E3 -348116.880}
SPL {X  -159.990, Y  +539.474, Z    +0.000, E1   +41.912, E3 -348130.407}
SPL {X  -159.990, Y  +544.879, Z    +0.000, E1   +41.899, E3 -348143.219}
SPL {X  -159.990, Y  +550.802, Z    +0.000, E1   +41.920, E3 -348157.200}
SPL {X  -159.990, Y  +556.952, Z    +0.000, E1   +41.911, E3 -348171.739}
SPL {X  -159.990, Y  +562.629, Z    +0.000, E1   +41.910, E3 -348185.157}
SPL {X  -159.990, Y  +567.682, Z    +0.000, E1   +41.901, E3 -348197.116}
SPL {X  -159.990, Y  +572.912, Z    +0.000, E1   +41.914, E3 -348209.464}
SPL {X  -159.990, Y  +578.863, Z    +0.000, E1   +41.918, E3 -348223.528}
SPL {X  -159.990, Y  +584.320, Z    +0.000, E1   +41.901, E3 -348236.474}
SPL {X  -159.990, Y  +589.217, Z    +0.000, E1   +41.901, E3 -348248.047}
SPL {X  -159.990, Y  +594.252, Z    +0.000, E1   +41.903, E3 -348259.962}
SPL {X  -159.990, Y  +598.793, Z    +0.000, E1   +41.896, E3 -348270.716}
SPL {X  -159.990, Y  +604.215, Z    +0.000, E1   +41.919, E3 -348283.496}
SPL {X  -159.990, Y  +610.545, Z    +0.000, E1   +41.917, E3 -348298.466}
SPL {X  -159.990, Y  +615.720, Z    +0.000, E1   +41.899, E3 -348310.726}
SPL {X  -159.990, Y  +621.417, Z    +0.000, E1   +41.931, E3 -348324.162}
SPL {X  -159.990, Y  +627.900, Z    +0.000, E1   +41.914, E3 -348339.502}
SPL {X  -159.990, Y  +634.411, Z    +0.000, E1   +41.931, E3 -348354.871}
SPL {X  -159.990, Y  +641.479, Z    +0.000, E1   +41.931, E3 -348371.588}
SPL {X  -159.990, Y  +647.782, Z    +0.000, E1   +41.914, E3 -348386.510}
SPL {X  -159.990, Y  +653.094, Z    +0.000, E1   +41.905, E3 -348399.088}
SPL {X  -159.990, Y  +657.893, Z    +0.000, E1   +41.899, E3 -348410.454}
SPL {X  -159.990, Y  +662.516, Z    +0.000, E1   +41.899, E3 -348421.385}
SPL {X  -159.990, Y  +668.411, Z    +0.000, E1   +41.929, E3 -348435.279}
SPL {X  -159.968, Y  +674.139, Z    +0.000, E1   +41.898, E3 -348448.883}
SPL {X  -159.817, Y  +678.937, Z    +0.000, E1   +41.879, E3 -348460.379}
SPL {X  -159.484, Y  +684.213, Z    +0.000, E1   +41.818, E3 -348473.215}
SPL {X  -159.007, Y  +689.209, Z    +0.000, E1   +41.732, E3 -348485.520}
SPL {X  -158.327, Y  +694.511, Z    +0.000, E1   +41.622, E3 -348498.771}
SPL {X  -157.480, Y  +699.729, Z    +0.000, E1   +41.453, E3 -348512.034}
SPL {X  -156.604, Y  +704.242, Z    +0.000, E1   +41.288, E3 -348523.642}
SPL {X  -155.831, Y  +707.744, Z    +0.000, E1   +41.132, E3 -348532.762}
SPL {X  -155.167, Y  +710.488, Z    +0.000, E1   +41.008, E3 -348539.940}
SPL {X  -154.232, Y  +714.035, Z    +0.000, E1   +40.861, E3 -348549.255}
SPL {X  -153.147, Y  +717.790, Z    +0.000, E1   +40.640, E3 -348559.273}
SPL {X  -151.881, Y  +721.788, Z    +0.000, E1   +40.435, E3 -348569.960}
SPL {X  -148.572, Y  +730.857, Z    +0.000, E1   +36.304, E3 -348626.169}
ENDSPLINE

SPLINE
SPL {X  -156.377, Y  +705.307, Z    +0.000, E1   +21.740, E3 -348680.417}
SPL {X  -159.301, Y  +686.331, Z    +0.000, E1   +11.648, E3 -348693.062}
SPL {X  -159.936, Y  +675.651, Z    +0.000, E1    +5.377, E3 -348696.778}
SPL {X  -159.990, Y  +670.142, Z    +0.000, E1    +1.740, E3 -348698.077}
SPL {X  -159.990, Y  +666.629, Z    +0.000, E1    -0.827, E3 -348698.727}
SPL {X  -159.990, Y  +662.407, Z    +0.000, E1    -4.406, E3 -348699.577}
SPL {X  -159.990, Y  +655.884, Z    +0.000, E1   -10.601, E3 -348701.442}
SPL {X  -159.990, Y  +646.242, Z    +0.000, E1   -19.956, E3 -348705.362}
SPL {X  -159.990, Y  +624.365, Z    +0.000, E1   -33.860, E3 -348723.263}
SPL {X  -159.990, Y  +615.596, Z    +0.000, E1   -36.980, E3 -348732.922}
SPL {X  -159.990, Y  +586.905, Z    +0.000, E1   -41.264, E3 -348779.948}
SPL {X  -159.990, Y  +581.111, Z    +0.000, E1   -41.245, E3 -348794.002}
SPL {X  -159.990, Y  +576.269, Z    +0.000, E1   -41.239, E3 -348805.729}
SPL {X  -159.990, Y  +571.714, Z    +0.000, E1   -41.240, E3 -348816.757}
SPL {X  -159.990, Y  +567.050, Z    +0.000, E1   -41.238, E3 -348828.044}
SPL {X  -159.990, Y  +561.959, Z    +0.000, E1   -41.251, E3 -348840.343}
SPL {X  -159.990, Y  +555.553, Z    +0.000, E1   -41.273, E3 -348855.811}
SPL {X  -159.990, Y  +549.897, Z    +0.000, E1   -41.240, E3 -348869.541}
SPL {X  -159.990, Y  +544.775, Z    +0.000, E1   -41.260, E3 -348881.916}
SPL {X  -159.990, Y  +538.952, Z    +0.000, E1   -41.247, E3 -348896.047}
SPL {X  -159.990, Y  +534.225, Z    +0.000, E1   -41.236, E3 -348907.480}
SPL {X  -159.990, Y  +529.136, Z    +0.000, E1   -41.262, E3 -348919.756}
SPL {X  -159.990, Y  +524.776, Z    +0.000, E1   -41.225, E3 -348930.369}
SPL {X  -159.990, Y  +521.454, Z    +0.000, E1   -41.236, E3 -348938.391}
SPL {X  -159.990, Y  +515.605, Z    +0.000, E1   -41.288, E3 -348952.431}
SPL {X  -159.990, Y  +509.898, Z    +0.000, E1   -41.246, E3 -348966.292}
SPL {X  -159.990, Y  +505.215, Z    +0.000, E1   -41.261, E3 -348977.608}
SPL {X  -159.990, Y  +500.102, Z    +0.000, E1   -41.251, E3 -348989.991}
SPL {X  -159.990, Y  +495.023, Z    +0.000, E1   -41.263, E3 -349002.240}
SPL {X  -159.990, Y  +479.011, Z    +0.000, E1   -45.740, E3 -349011.622}
SPL {X  -159.990, Y  +471.379, Z    +0.000, E1   -46.435, E3 -349023.237}
SPL {X  -159.990, Y  +466.895, Z    +0.000, E1   -45.533, E3 -349037.642}
SPL {X  -159.990, Y  +462.409, Z    +0.000, E1   -44.664, E3 -349052.417}
SPL {X  -159.990, Y  +458.229, Z    +0.000, E1   -43.579, E3 -349067.899}
SPL {X  -159.990, Y  +453.434, Z    +0.000, E1   -43.227, E3 -349080.674}
SPL {X  -159.990, Y  +448.702, Z    +0.000, E1   -43.218, E3 -349091.395}
SPL {X  -159.990, Y  +444.476, Z    +0.000, E1   -43.219, E3 -349100.934}
SPL {X  -159.990, Y  +440.246, Z    +0.000, E1   -43.217, E3 -349110.491}
SPL {X  -159.990, Y  +434.411, Z    +0.000, E1   -43.246, E3 -349123.622}
SPL {X  -159.990, Y  +429.216, Z    +0.000, E1   -43.210, E3 -349135.394}
SPL {X  -159.990, Y  +424.433, Z    +0.000, E1   -43.237, E3 -349146.142}
SPL {X  -159.990, Y  +419.466, Z    +0.000, E1   -43.217, E3 -349157.382}
SPL {X  -159.990, Y  +414.585, Z    +0.000, E1   -43.233, E3 -349168.373}
SPL {X  -159.990, Y  +409.927, Z    +0.000, E1   -43.217, E3 -349178.905}
SPL {X  -159.990, Y  +405.428, Z    +0.000, E1   -43.230, E3 -349189.063}
SPL {X  -159.990, Y  +401.033, Z    +0.000, E1   -43.209, E3 -349199.018}
SPL {X  -159.990, Y  +396.968, Z    +0.000, E1   -43.221, E3 -349208.176}
SPL {X  -159.990, Y  +392.163, Z    +0.000, E1   -43.223, E3 -349219.018}
SPL {X  -159.990, Y  +387.342, Z    +0.000, E1   -43.224, E3 -349229.895}
SPL {X  -159.990, Y  +382.548, Z    +0.000, E1   -43.224, E3 -349240.718}
SPL {X  -159.922, Y  +377.835, Z    +0.000, E1   -43.211, E3 -349251.435}
SPL {X  -159.712, Y  +373.072, Z    +0.000, E1   -43.177, E3 -349262.401}
SPL {X  -159.289, Y  +367.537, Z    +0.000, E1   -43.118, E3 -349275.312}
SPL {X  -158.730, Y  +362.464, Z    +0.000, E1   -43.003, E3 -349287.344}
SPL {X  -158.182, Y  +358.518, Z    +0.000, E1   -42.902, E3 -349296.823}
SPL {X  -157.507, Y  +354.423, Z    +0.000, E1   -42.786, E3 -349306.768}
SPL {X  -156.676, Y  +350.104, Z    +0.000, E1   -42.637, E3 -349317.373}
SPL {X  -155.807, Y  +346.154, Z    +0.000, E1   -42.470, E3 -349327.201}
SPL {X  -154.777, Y  +341.993, Z    +0.000, E1   -42.302, E3 -349337.626}
SPL {X  -153.585, Y  +337.686, Z    +0.000, E1   -42.062, E3 -349348.601}
SPL {X  -152.412, Y  +333.846, Z    +0.000, E1   -41.856, E3 -349358.444}
SPL {X  -151.009, Y  +329.651, Z    +0.000, E1   -41.581, E3 -349369.343}
SPL {X  -148.356, Y  +322.607, Z    +0.000, E1   -36.121, E3 -349429.819}
ENDSPLINE

SPLINE
SPL {X  -156.487, Y  +349.204, Z    +0.000, E1   -21.338, E3 -349484.945}
SPL {X  -159.136, Y  +365.992, Z    +0.000, E1   -12.463, E3 -349495.703}
SPL {X  -159.799, Y  +374.694, Z    +0.000, E1    -7.504, E3 -349498.807}
SPL {X  -159.976, Y  +380.404, Z    +0.000, E1    -3.959, E3 -349500.340}
SPL {X  -159.990, Y  +384.773, Z    +0.000, E1    -1.003, E3 -349501.235}
SPL {X  -159.990, Y  +387.968, Z    +0.000, E1    +1.448, E3 -349501.803}
SPL {X  -159.990, Y  +391.397, Z    +0.000, E1    +4.422, E3 -349502.427}
SPL {X  -159.990, Y  +395.864, Z    +0.000, E1    +8.712, E3 -349503.515}
SPL {X  -159.990, Y  +401.273, Z    +0.000, E1   +14.176, E3 -349505.243}
SPL {X  -159.990, Y  +409.369, Z    +0.000, E1   +21.807, E3 -349509.035}
SPL {X  -159.990, Y  +436.107, Z    +0.000, E1   +36.921, E3 -349531.960}
SPL {X  -159.990, Y  +465.724, Z    +0.000, E1   +41.883, E3 -349576.758}
SPL {X  -159.990, Y  +470.837, Z    +0.000, E1   +41.927, E3 -349588.772}
SPL {X  -159.990, Y  +477.498, Z    +0.000, E1   +41.916, E3 -349604.548}
SPL {X  -159.990, Y  +484.724, Z    +0.000, E1   +41.943, E3 -349621.586}
SPL {X  -159.990, Y  +492.944, Z    +0.000, E1   +41.952, E3 -349641.005}
SPL {X  -159.990, Y  +499.538, Z    +0.000, E1   +41.904, E3 -349656.664}
SPL {X  -159.990, Y  +505.259, Z    +0.000, E1   +41.922, E3 -349670.163}
SPL {X  -159.990, Y  +511.862, Z    +0.000, E1   +41.927, E3 -349685.773}
SPL {X  -159.990, Y  +517.450, Z    +0.000, E1   +41.901, E3 -349699.021}
SPL {X  -159.990, Y  +523.027, Z    +0.000, E1   +41.926, E3 -349712.165}
SPL {X  -159.990, Y  +528.611, Z    +0.000, E1   +41.900, E3 -349725.420}
SPL {X  -159.990, Y  +533.758, Z    +0.000, E1   +41.910, E3 -349737.570}
SPL {X  -159.990, Y  +539.474, Z    +0.000, E1   +41.912, E3 -349751.097}
SPL {X  -159.990, Y  +544.879, Z    +0.000, E1   +41.899, E3 -349763.908}
SPL {X  -159.990, Y  +550.802, Z    +0.000, E1   +41.920, E3 -349777.890}
SPL {X  -159.990, Y  +556.952, Z    +0.000, E1   +41.911, E3 -349792.429}
SPL {X  -159.990, Y  +562.629, Z    +0.000, E1   +41.910, E3 -349805.847}
SPL {X  -159.990, Y  +567.682, Z    +0.000, E1   +41.901, E3 -349817.806}
SPL {X  -159.990, Y  +572.912, Z    +0.000, E1   +41.914, E3 -349830.153}
SPL {X  -159.990, Y  +578.863, Z    +0.000, E1   +41.918, E3 -349844.217}
SPL {X  -159.990, Y  +584.320, Z    +0.000, E1   +41.901, E3 -349857.164}
SPL {X  -159.990, Y  +589.217, Z    +0.000, E1   +41.901, E3 -349868.737}
SPL {X  -159.990, Y  +594.252, Z    +0.000, E1   +41.903, E3 -349880.651}
SPL {X  -159.990, Y  +598.793, Z    +0.000, E1   +41.896, E3 -349891.405}
SPL {X  -159.990, Y  +604.215, Z    +0.000, E1   +41.919, E3 -349904.186}
SPL {X  -159.990, Y  +610.545, Z    +0.000, E1   +41.917, E3 -349919.155}
SPL {X  -159.990, Y  +615.720, Z    +0.000, E1   +41.899, E3 -349931.415}
SPL {X  -159.990, Y  +620.005, Z    +0.000, E1   +41.900, E3 -349941.548}
SPL {X  -159.990, Y  +624.919, Z    +0.000, E1   +41.912, E3 -349953.156}
SPL {X  -159.990, Y  +630.816, Z    +0.000, E1   +41.915, E3 -349967.085}
SPL {X  -159.990, Y  +637.009, Z    +0.000, E1   +41.925, E3 -349981.710}
SPL {X  -159.990, Y  +642.624, Z    +0.000, E1   +41.901, E3 -349995.031}
SPL {X  -159.990, Y  +647.782, Z    +0.000, E1   +41.914, E3 -350007.199}
SPL {X  -159.990, Y  +653.094, Z    +0.000, E1   +41.905, E3 -350019.778}
SPL {X  -159.990, Y  +657.893, Z    +0.000, E1   +41.899, E3 -350031.143}
SPL {X  -159.990, Y  +662.516, Z    +0.000, E1   +41.899, E3 -350042.075}
SPL {X  -159.990, Y  +668.411, Z    +0.000, E1   +41.929, E3 -350055.968}
SPL {X  -159.968, Y  +674.139, Z    +0.000, E1   +41.898, E3 -350069.572}
SPL {X  -159.817, Y  +678.937, Z    +0.000, E1   +41.879, E3 -350081.068}
SPL {X  -159.484, Y  +684.213, Z    +0.000, E1   +41.818, E3 -350093.905}
SPL {X  -159.007, Y  +689.209, Z    +0.000, E1   +41.732, E3 -350106.209}
SPL {X  -158.327, Y  +694.511, Z    +0.000, E1   +41.622, E3 -350119.460}
SPL {X  -157.480, Y  +699.729, Z    +0.000, E1   +41.453, E3 -350132.723}
SPL {X  -156.604, Y  +704.242, Z    +0.000, E1   +41.288, E3 -350144.332}
SPL {X  -155.514, Y  +709.078, Z    +0.000, E1   +41.107, E3 -350156.886}
SPL {X  -154.232, Y  +714.035, Z    +0.000, E1   +40.861, E3 -350169.945}
SPL {X  -153.147, Y  +717.790, Z    +0.000, E1   +40.640, E3 -350179.963}
SPL {X  -151.881, Y  +721.788, Z    +0.000, E1   +40.435, E3 -350190.649}
SPL {X  -148.572, Y  +730.857, Z    +0.000, E1   +36.304, E3 -350246.858}
ENDSPLINE

SPLINE
SPL {X  -156.377, Y  +705.307, Z    +0.000, E1   +21.740, E3 -350301.107}
SPL {X  -159.301, Y  +686.331, Z    +0.000, E1   +11.648, E3 -350313.752}
SPL {X  -159.936, Y  +675.651, Z    +0.000, E1    +5.377, E3 -350317.467}
SPL {X  -159.990, Y  +670.142, Z    +0.000, E1    +1.740, E3 -350318.767}
SPL {X  -159.990, Y  +666.629, Z    +0.000, E1    -0.827, E3 -350319.416}
SPL {X  -159.990, Y  +662.407, Z    +0.000, E1    -4.406, E3 -350320.267}
SPL {X  -159.990, Y  +657.382, Z    +0.000, E1    -9.217, E3 -350321.649}
SPL {X  -159.990, Y  +653.255, Z    +0.000, E1   -13.347, E3 -350322.978}
SPL {X  -159.990, Y  +643.833, Z    +0.000, E1   -21.883, E3 -350327.761}
SPL {X  -159.990, Y  +617.235, Z    +0.000, E1   -36.481, E3 -350351.661}
SPL {X  -159.990, Y  +586.905, Z    +0.000, E1   -41.264, E3 -350400.638}
SPL {X  -159.990, Y  +581.111, Z    +0.000, E1   -41.245, E3 -350414.692}
SPL {X  -159.990, Y  +576.269, Z    +0.000, E1   -41.239, E3 -350426.419}
SPL {X  -159.990, Y  +571.714, Z    +0.000, E1   -41.240, E3 -350437.447}
SPL {X  -159.990, Y  +567.050, Z    +0.000, E1   -41.238, E3 -350448.734}
SPL {X  -159.990, Y  +561.959, Z    +0.000, E1   -41.251, E3 -350461.032}
SPL {X  -159.990, Y  +557.719, Z    +0.000, E1   -41.226, E3 -350471.335}
SPL {X  -159.990, Y  +554.148, Z    +0.000, E1   -41.237, E3 -350479.950}
SPL {X  -159.990, Y  +548.812, Z    +0.000, E1   -41.263, E3 -350492.825}
SPL {X  -159.990, Y  +543.804, Z    +0.000, E1   -41.237, E3 -350504.989}
SPL {X  -159.990, Y  +538.952, Z    +0.000, E1   -41.247, E3 -350516.737}
SPL {X  -159.990, Y  +534.225, Z    +0.000, E1   -41.236, E3 -350528.170}
SPL {X  -159.990, Y  +529.136, Z    +0.000, E1   -41.262, E3 -350540.446}
SPL {X  -159.990, Y  +522.690, Z    +0.000, E1   -41.265, E3 -350556.045}
SPL {X  -159.990, Y  +516.698, Z    +0.000, E1   -41.259, E3 -350570.520}
SPL {X  -159.990, Y  +510.896, Z    +0.000, E1   -41.267, E3 -350584.537}
SPL {X  -159.990, Y  +505.215, Z    +0.000, E1   -41.261, E3 -350598.297}
SPL {X  -159.990, Y  +500.102, Z    +0.000, E1   -41.251, E3 -350610.681}
SPL {X  -159.990, Y  +495.023, Z    +0.000, E1   -41.263, E3 -350622.930}
SPL {X  -159.990, Y  +479.011, Z    +0.000, E1   -45.740, E3 -350632.312}
SPL {X  -159.990, Y  +471.379, Z    +0.000, E1   -46.435, E3 -350643.927}
SPL {X  -159.990, Y  +465.881, Z    +0.000, E1   -45.385, E3 -350661.530}
SPL {X  -159.990, Y  +461.571, Z    +0.000, E1   -44.440, E3 -350676.055}
SPL {X  -159.990, Y  +458.229, Z    +0.000, E1   -43.579, E3 -350688.589}
SPL {X  -159.990, Y  +453.434, Z    +0.000, E1   -43.227, E3 -350701.363}
SPL {X  -159.990, Y  +448.702, Z    +0.000, E1   -43.218, E3 -350712.085}
SPL {X  -159.990, Y  +444.476, Z    +0.000, E1   -43.219, E3 -350721.623}
SPL {X  -159.990, Y  +440.246, Z    +0.000, E1   -43.217, E3 -350731.181}
SPL {X  -159.990, Y  +434.411, Z    +0.000, E1   -43.246, E3 -350744.311}
SPL {X  -159.990, Y  +429.216, Z    +0.000, E1   -43.210, E3 -350756.084}
SPL {X  -159.990, Y  +424.433, Z    +0.000, E1   -43.237, E3 -350766.832}
SPL {X  -159.990, Y  +419.466, Z    +0.000, E1   -43.217, E3 -350778.071}
SPL {X  -159.990, Y  +414.585, Z    +0.000, E1   -43.233, E3 -350789.063}
SPL {X  -159.990, Y  +409.927, Z    +0.000, E1   -43.217, E3 -350799.595}
SPL {X  -159.990, Y  +405.428, Z    +0.000, E1   -43.230, E3 -350809.753}
SPL {X  -159.990, Y  +398.518, Z    +0.000, E1   -43.261, E3 -350825.307}
SPL {X  -159.990, Y  +392.163, Z    +0.000, E1   -43.223, E3 -350839.707}
SPL {X  -159.990, Y  +387.342, Z    +0.000, E1   -43.224, E3 -350850.585}
SPL {X  -159.990, Y  +382.548, Z    +0.000, E1   -43.224, E3 -350861.408}
SPL {X  -159.922, Y  +377.835, Z    +0.000, E1   -43.211, E3 -350872.124}
SPL {X  -159.712, Y  +373.072, Z    +0.000, E1   -43.177, E3 -350883.090}
SPL {X  -159.289, Y  +367.537, Z    +0.000, E1   -43.118, E3 -350896.002}
SPL {X  -158.730, Y  +362.464, Z    +0.000, E1   -43.003, E3 -350908.034}
SPL {X  -158.182, Y  +358.518, Z    +0.000, E1   -42.902, E3 -350917.513}
SPL {X  -157.507, Y  +354.423, Z    +0.000, E1   -42.786, E3 -350927.458}
SPL {X  -156.676, Y  +350.104, Z    +0.000, E1   -42.637, E3 -350938.063}
SPL {X  -155.807, Y  +346.154, Z    +0.000, E1   -42.470, E3 -350947.890}
SPL {X  -154.777, Y  +341.993, Z    +0.000, E1   -42.302, E3 -350958.315}
SPL {X  -153.585, Y  +337.686, Z    +0.000, E1   -42.062, E3 -350969.291}
SPL {X  -152.412, Y  +333.846, Z    +0.000, E1   -41.856, E3 -350979.133}
SPL {X  -151.009, Y  +329.651, Z    +0.000, E1   -41.581, E3 -350990.033}
SPL {X  -148.356, Y  +322.607, Z    +0.000, E1   -36.121, E3 -351050.509}
ENDSPLINE

SPLINE
SPL {X  -156.487, Y  +349.204, Z    +0.000, E1   -21.338, E3 -351105.635}
SPL {X  -159.136, Y  +365.992, Z    +0.000, E1   -12.463, E3 -351116.393}
SPL {X  -159.799, Y  +374.694, Z    +0.000, E1    -7.504, E3 -351119.497}
SPL {X  -159.976, Y  +380.404, Z    +0.000, E1    -3.959, E3 -351121.030}
SPL {X  -159.990, Y  +384.773, Z    +0.000, E1    -1.003, E3 -351121.924}
SPL {X  -159.990, Y  +387.968, Z    +0.000, E1    +1.448, E3 -351122.493}
SPL {X  -159.990, Y  +391.397, Z    +0.000, E1    +4.422, E3 -351123.117}
SPL {X  -159.990, Y  +395.864, Z    +0.000, E1    +8.712, E3 -351124.205}
SPL {X  -159.990, Y  +401.273, Z    +0.000, E1   +14.176, E3 -351125.932}
SPL {X  -159.990, Y  +409.369, Z    +0.000, E1   +21.807, E3 -351129.724}
SPL {X  -159.990, Y  +436.107, Z    +0.000, E1   +36.921, E3 -351152.650}
SPL {X  -159.990, Y  +468.567, Z    +0.000, E1   +41.922, E3 -351204.097}
SPL {X  -159.990, Y  +474.616, Z    +0.000, E1   +41.909, E3 -351218.426}
SPL {X  -159.990, Y  +478.952, Z    +0.000, E1   +41.885, E3 -351228.724}
SPL {X  -159.990, Y  +484.724, Z    +0.000, E1   +41.943, E3 -351242.276}
SPL {X  -159.990, Y  +492.944, Z    +0.000, E1   +41.952, E3 -351261.695}
SPL {X  -159.990, Y  +499.538, Z    +0.000, E1   +41.904, E3 -351277.354}
SPL {X  -159.990, Y  +504.097, Z    +0.000, E1   +41.897, E3 -351288.142}
SPL {X  -159.990, Y  +509.413, Z    +0.000, E1   +41.921, E3 -351300.677}
SPL {X  -159.990, Y  +516.193, Z    +0.000, E1   +41.932, E3 -351316.693}
SPL {X  -159.990, Y  +523.027, Z    +0.000, E1   +41.926, E3 -351332.855}
SPL {X  -159.990, Y  +528.611, Z    +0.000, E1   +41.900, E3 -351346.110}
SPL {X  -159.990, Y  +533.758, Z    +0.000, E1   +41.910, E3 -351358.259}
SPL {X  -159.990, Y  +539.474, Z    +0.000, E1   +41.912, E3 -351371.787}
SPL {X  -159.990, Y  +544.879, Z    +0.000, E1   +41.899, E3 -351384.598}
SPL {X  -159.990, Y  +550.802, Z    +0.000, E1   +41.920, E3 -351398.579}
SPL {X  -159.990, Y  +556.952, Z    +0.000, E1   +41.911, E3 -351413.119}
SPL {X  -159.990, Y  +562.629, Z    +0.000, E1   +41.910, E3 -351426.537}
SPL {X  -159.990, Y  +567.682, Z    +0.000, E1   +41.901, E3 -351438.496}
SPL {X  -159.990, Y  +572.912, Z    +0.000, E1   +41.914, E3 -351450.843}
SPL {X  -159.990, Y  +578.863, Z    +0.000, E1   +41.918, E3 -351464.907}
SPL {X  -159.990, Y  +584.320, Z    +0.000, E1   +41.901, E3 -351477.854}
SPL {X  -159.990, Y  +589.217, Z    +0.000, E1   +41.901, E3 -351489.426}
SPL {X  -159.990, Y  +594.252, Z    +0.000, E1   +41.903, E3 -351501.341}
SPL {X  -159.990, Y  +600.237, Z    +0.000, E1   +41.928, E3 -351515.459}
SPL {X  -159.990, Y  +607.478, Z    +0.000, E1   +41.933, E3 -351532.567}
SPL {X  -159.990, Y  +614.570, Z    +0.000, E1   +41.926, E3 -351549.348}
SPL {X  -159.990, Y  +621.417, Z    +0.000, E1   +41.931, E3 -351565.542}
SPL {X  -159.990, Y  +627.900, Z    +0.000, E1   +41.914, E3 -351580.881}
SPL {X  -159.990, Y  +632.270, Z    +0.000, E1   +41.887, E3 -351591.257}
SPL {X  -159.990, Y  +637.009, Z    +0.000, E1   +41.925, E3 -351602.400}
SPL {X  -159.990, Y  +642.624, Z    +0.000, E1   +41.901, E3 -351615.721}
SPL {X  -159.990, Y  +647.782, Z    +0.000, E1   +41.914, E3 -351627.889}
SPL {X  -159.990, Y  +653.094, Z    +0.000, E1   +41.905, E3 -351640.467}
SPL {X  -159.990, Y  +657.893, Z    +0.000, E1   +41.899, E3 -351651.833}
SPL {X  -159.990, Y  +662.516, Z    +0.000, E1   +41.899, E3 -351662.764}
SPL {X  -159.990, Y  +668.411, Z    +0.000, E1   +41.929, E3 -351676.658}
SPL {X  -159.968, Y  +674.139, Z    +0.000, E1   +41.898, E3 -351690.262}
SPL {X  -159.817, Y  +678.937, Z    +0.000, E1   +41.879, E3 -351701.758}
SPL {X  -159.484, Y  +684.213, Z    +0.000, E1   +41.818, E3 -351714.594}
SPL {X  -159.007, Y  +689.209, Z    +0.000, E1   +41.732, E3 -351726.899}
SPL {X  -158.327, Y  +694.511, Z    +0.000, E1   +41.622, E3 -351740.150}
SPL {X  -157.480, Y  +699.729, Z    +0.000, E1   +41.453, E3 -351753.413}
SPL {X  -156.604, Y  +704.242, Z    +0.000, E1   +41.288, E3 -351765.022}
SPL {X  -155.831, Y  +707.744, Z    +0.000, E1   +41.132, E3 -351774.142}
SPL {X  -155.167, Y  +710.488, Z    +0.000, E1   +41.008, E3 -351781.320}
SPL {X  -154.232, Y  +714.035, Z    +0.000, E1   +40.861, E3 -351790.634}
SPL {X  -153.147, Y  +717.790, Z    +0.000, E1   +40.640, E3 -351800.653}
SPL {X  -151.881, Y  +721.788, Z    +0.000, E1   +40.435, E3 -351811.339}
SPL {X  -148.572, Y  +730.857, Z    +0.000, E1   +36.304, E3 -351867.548}
ENDSPLINE

SPLINE
SPL {X  -156.377, Y  +705.307, Z    +0.000, E1   +21.740, E3 -351921.797}
SPL {X  -159.301, Y  +686.331, Z    +0.000, E1   +11.648, E3 -351934.441}
SPL {X  -159.936, Y  +675.651, Z    +0.000, E1    +5.377, E3 -351938.157}
SPL {X  -159.990, Y  +670.142, Z    +0.000, E1    +1.740, E3 -351939.456}
SPL {X  -159.990, Y  +666.629, Z    +0.000, E1    -0.827, E3 -351940.106}
SPL {X  -159.990, Y  +662.407, Z    +0.000, E1    -4.406, E3 -351940.956}
SPL {X  -159.990, Y  +657.382, Z    +0.000, E1    -9.217, E3 -351942.338}
SPL {X  -159.990, Y  +653.255, Z    +0.000, E1   -13.347, E3 -351943.667}
SPL {X  -159.990, Y  +646.242, Z    +0.000, E1   -19.956, E3 -351946.741}
SPL {X  -159.990, Y  +624.365, Z    +0.000, E1   -33.860, E3 -351964.642}
SPL {X  -159.990, Y  +615.596, Z    +0.000, E1   -36.980, E3 -351974.301}
SPL {X  -159.990, Y  +586.905, Z    +0.000, E1   -41.264, E3 -352021.327}
SPL {X  -159.990, Y  +581.111, Z    +0.000, E1   -41.245, E3 -352035.381}
SPL {X  -159.990, Y  +576.269, Z    +0.000, E1   -41.239, E3 -352047.109}
SPL {X  -159.990, Y  +571.714, Z    +0.000, E1   -41.240, E3 -352058.137}
SPL {X  -159.990, Y  +567.050, Z    +0.000, E1   -41.238, E3 -352069.424}
SPL {X  -159.990, Y  +561.959, Z    +0.000, E1   -41.251, E3 -352081.722}
SPL {X  -159.990, Y  +555.553, Z    +0.000, E1   -41.273, E3 -352097.190}
SPL {X  -159.990, Y  +548.812, Z    +0.000, E1   -41.263, E3 -352113.514}
SPL {X  -159.990, Y  +543.804, Z    +0.000, E1   -41.237, E3 -352125.679}
SPL {X  -159.990, Y  +538.952, Z    +0.000, E1   -41.247, E3 -352137.426}
SPL {X  -159.990, Y  +534.225, Z    +0.000, E1   -41.236, E3 -352148.859}
SPL {X  -159.990, Y  +529.136, Z    +0.000, E1   -41.262, E3 -352161.135}
SPL {X  -159.990, Y  +522.690, Z    +0.000, E1   -41.265, E3 -352176.735}
SPL {X  -159.990, Y  +515.605, Z    +0.000, E1   -41.288, E3 -352193.810}
SPL {X  -159.990, Y  +509.898, Z    +0.000, E1   -41.246, E3 -352207.671}
SPL {X  -159.990, Y  +505.215, Z    +0.000, E1   -41.261, E3 -352218.987}
SPL {X  -159.990, Y  +500.102, Z    +0.000, E1   -41.251, E3 -352231.370}
SPL {X  -159.990, Y  +495.023, Z    +0.000, E1   -41.263, E3 -352243.619}
SPL {X  -159.990, Y  +479.011, Z    +0.000, E1   -45.740, E3 -352253.001}
SPL {X  -159.990, Y  +471.379, Z    +0.000, E1   -46.435, E3 -352264.617}
SPL {X  -159.990, Y  +465.881, Z    +0.000, E1   -45.385, E3 -352282.219}
SPL {X  -159.990, Y  +461.571, Z    +0.000, E1   -44.440, E3 -352296.745}
SPL {X  -159.990, Y  +458.229, Z    +0.000, E1   -43.579, E3 -352309.278}
SPL {X  -159.990, Y  +453.434, Z    +0.000, E1   -43.227, E3 -352322.053}
SPL {X  -159.990, Y  +448.702, Z    +0.000, E1   -43.218, E3 -352332.775}
SPL {X  -159.990, Y  +442.224, Z    +0.000, E1   -43.270, E3 -352347.325}
SPL {X  -159.990, Y  +434.411, Z    +0.000, E1   -43.246, E3 -352365.001}
SPL {X  -159.990, Y  +429.216, Z    +0.000, E1   -43.210, E3 -352376.773}
SPL {X  -159.990, Y  +424.433, Z    +0.000, E1   -43.237, E3 -352387.521}
SPL {X  -159.990, Y  +419.466, Z    +0.000, E1   -43.217, E3 -352398.761}
SPL {X  -159.990, Y  +414.585, Z    +0.000, E1   -43.233, E3 -352409.753}
SPL {X  -159.990, Y  +409.927, Z    +0.000, E1   -43.217, E3 -352420.284}
SPL {X  -159.990, Y  +405.428, Z    +0.000, E1   -43.230, E3 -352430.443}
SPL {X  -159.990, Y  +398.518, Z    +0.000, E1   -43.261, E3 -352445.997}
SPL {X  -159.990, Y  +392.163, Z    +0.000, E1   -43.223, E3 -352460.397}
SPL {X  -159.990, Y  +387.342, Z    +0.000, E1   -43.224, E3 -352471.275}
SPL {X  -159.990, Y  +382.548, Z    +0.000, E1   -43.224, E3 -352482.097}
SPL {X  -159.922, Y  +377.835, Z    +0.000, E1   -43.211, E3 -352492.814}
SPL {X  -159.712, Y  +373.072, Z    +0.000, E1   -43.177, E3 -352503.780}
SPL {X  -159.289, Y  +367.537, Z    +0.000, E1   -43.118, E3 -352516.692}
SPL {X  -158.730, Y  +362.464, Z    +0.000, E1   -43.003, E3 -352528.724}
SPL {X  -158.182, Y  +358.518, Z    +0.000, E1   -42.902, E3 -352538.202}
SPL {X  -157.507, Y  +354.423, Z    +0.000, E1   -42.786, E3 -352548.148}
SPL {X  -156.676, Y  +350.104, Z    +0.000, E1   -42.637, E3 -352558.753}
SPL {X  -155.807, Y  +346.154, Z    +0.000, E1   -42.470, E3 -352568.580}
SPL {X  -154.777, Y  +341.993, Z    +0.000, E1   -42.302, E3 -352579.005}
SPL {X  -153.585, Y  +337.686, Z    +0.000, E1   -42.062, E3 -352589.980}
SPL {X  -152.412, Y  +333.846, Z    +0.000, E1   -41.856, E3 -352599.823}
SPL {X  -151.009, Y  +329.651, Z    +0.000, E1   -41.581, E3 -352610.723}
SPL {X  -148.356, Y  +322.607, Z    +0.000, E1   -36.121, E3 -352671.198}
ENDSPLINE

SPLINE
SPL {X  -156.487, Y  +349.204, Z    +0.000, E1   -21.338, E3 -352726.324}
SPL {X  -159.136, Y  +365.992, Z    +0.000, E1   -12.463, E3 -352737.083}
SPL {X  -159.799, Y  +374.694, Z    +0.000, E1    -7.504, E3 -352740.187}
SPL {X  -159.976, Y  +380.404, Z    +0.000, E1    -3.959, E3 -352741.720}
SPL {X  -159.990, Y  +384.773, Z    +0.000, E1    -1.003, E3 -352742.614}
SPL {X  -159.990, Y  +387.968, Z    +0.000, E1    +1.448, E3 -352743.182}
SPL {X  -159.990, Y  +391.397, Z    +0.000, E1    +4.422, E3 -352743.806}
SPL {X  -159.990, Y  +395.864, Z    +0.000, E1    +8.712, E3 -352744.895}
SPL {X  -159.990, Y  +401.273, Z    +0.000, E1   +14.176, E3 -352746.622}
SPL {X  -159.990, Y  +409.369, Z    +0.000, E1   +21.807, E3 -352750.414}
SPL {X  -159.990, Y  +436.107, Z    +0.000, E1   +36.921, E3 -352773.339}
SPL {X  -159.990, Y  +465.724, Z    +0.000, E1   +41.883, E3 -352818.137}
SPL {X  -159.990, Y  +470.837, Z    +0.000, E1   +41.927, E3 -352830.152}
SPL {X  -159.990, Y  +477.498, Z    +0.000, E1   +41.916, E3 -352845.927}
SPL {X  -159.990, Y  +484.724, Z    +0.000, E1   +41.943, E3 -352862.965}
SPL {X  -159.990, Y  +492.944, Z    +0.000, E1   +41.952, E3 -352882.385}
SPL {X  -159.990, Y  +499.538, Z    +0.000, E1   +41.904, E3 -352898.043}
SPL {X  -159.990, Y  +505.259, Z    +0.000, E1   +41.922, E3 -352911.542}
SPL {X  -159.990, Y  +511.862, Z    +0.000, E1   +41.927, E3 -352927.153}
SPL {X  -159.990, Y  +517.450, Z    +0.000, E1   +41.901, E3 -352940.400}
SPL {X  -159.990, Y  +523.027, Z    +0.000, E1   +41.926, E3 -352953.544}
SPL {X  -159.990, Y  +528.611, Z    +0.000, E1   +41.900, E3 -352966.800}
SPL {X  -159.990, Y  +533.758, Z    +0.000, E1   +41.910, E3 -352978.949}
SPL {X  -159.990, Y  +539.474, Z    +0.000, E1   +41.912, E3 -352992.476}
SPL {X  -159.990, Y  +544.879, Z    +0.000, E1   +41.899, E3 -353005.288}
SPL {X  -159.990, Y  +550.802, Z    +0.000, E1   +41.920, E3 -353019.269}
SPL {X  -159.990, Y  +556.952, Z    +0.000, E1   +41.911, E3 -353033.808}
SPL {X  -159.990, Y  +562.629, Z    +0.000, E1   +41.910, E3 -353047.226}
SPL {X  -159.990, Y  +567.682, Z    +0.000, E1   +41.901, E3 -353059.185}
SPL {X  -159.990, Y  +572.912, Z    +0.000, E1   +41.914, E3 -353071.533}
SPL {X  -159.990, Y  +578.863, Z    +0.000, E1   +41.918, E3 -353085.597}
SPL {X  -159.990, Y  +584.320, Z    +0.000, E1   +41.901, E3 -353098.543}
SPL {X  -159.990, Y  +589.217, Z    +0.000, E1   +41.901, E3 -353110.116}
SPL {X  -159.990, Y  +594.252, Z    +0.000, E1   +41.903, E3 -353122.031}
SPL {X  -159.990, Y  +598.793, Z    +0.000, E1   +41.896, E3 -353132.785}
SPL {X  -159.990, Y  +604.215, Z    +0.000, E1   +41.919, E3 -353145.565}
SPL {X  -159.990, Y  +610.545, Z    +0.000, E1   +41.917, E3 -353160.535}
SPL {X  -159.990, Y  +615.720, Z    +0.000, E1   +41.899, E3 -353172.795}
SPL {X  -159.990, Y  +621.417, Z    +0.000, E1   +41.931, E3 -353186.231}
SPL {X  -159.990, Y  +627.900, Z    +0.000, E1   +41.914, E3 -353201.571}
SPL {X  -159.990, Y  +634.411, Z    +0.000, E1   +41.931, E3 -353216.940}
SPL {X  -159.990, Y  +641.479, Z    +0.000, E1   +41.931, E3 -353233.657}
SPL {X  -159.990, Y  +647.782, Z    +0.000, E1   +41.914, E3 -353248.579}
SPL {X  -159.990, Y  +653.094, Z    +0.000, E1   +41.905, E3 -353261.157}
SPL {X  -159.990, Y  +657.893, Z    +0.000, E1   +41.899, E3 -353272.523}
SPL {X  -159.990, Y  +662.516, Z    +0.000, E1   +41.899, E3 -353283.454}
SPL {X  -159.990, Y  +668.411, Z    +0.000, E1   +41.929, E3 -353297.348}
SPL {X  -159.968, Y  +674.139, Z    +0.000, E1   +41.898, E3 -353310.952}
SPL {X  -159.817, Y  +678.937, Z    +0.000, E1   +41.879, E3 -353322.448}
SPL {X  -159.484, Y  +684.213, Z    +0.000, E1   +41.818, E3 -353335.284}
SPL {X  -159.007, Y  +689.209, Z    +0.000, E1   +41.732, E3 -353347.589}
SPL {X  -158.327, Y  +694.511, Z    +0.000, E1   +41.622, E3 -353360.840}
SPL {X  -157.480, Y  +699.729, Z    +0.000, E1   +41.453, E3 -353374.103}
SPL {X  -156.604, Y  +704.242, Z    +0.000, E1   +41.288, E3 -353385.711}
SPL {X  -155.831, Y  +707.744, Z    +0.000, E1   +41.132, E3 -353394.831}
SPL {X  -155.167, Y  +710.488, Z    +0.000, E1   +41.008, E3 -353402.009}
SPL {X  -154.232, Y  +714.035, Z    +0.000, E1   +40.861, E3 -353411.324}
SPL {X  -153.147, Y  +717.790, Z    +0.000, E1   +40.640, E3 -353421.342}
SPL {X  -151.881, Y  +721.788, Z    +0.000, E1   +40.435, E3 -353432.029}
SPL {X  -148.572, Y  +730.857, Z    +0.000, E1   +36.304, E3 -353488.238}
ENDSPLINE

SPLINE
SPL {X  -156.377, Y  +705.307, Z    +0.000, E1   +21.740, E3 -353542.486}
SPL {X  -159.301, Y  +686.331, Z    +0.000, E1   +11.648, E3 -353555.131}
SPL {X  -159.936, Y  +675.651, Z    +0.000, E1    +5.377, E3 -353558.847}
SPL {X  -159.990, Y  +670.142, Z    +0.000, E1    +1.740, E3 -353560.146}
SPL {X  -159.990, Y  +666.629, Z    +0.000, E1    -0.827, E3 -353560.796}
SPL {X  -159.990, Y  +662.407, Z    +0.000, E1    -4.406, E3 -353561.646}
SPL {X  -159.990, Y  +655.884, Z    +0.000, E1   -10.601, E3 -353563.511}
SPL {X  -159.990, Y  +646.242, Z    +0.000, E1   -19.956, E3 -353567.431}
SPL {X  -159.990, Y  +624.365, Z    +0.000, E1   -33.860, E3 -353585.332}
SPL {X  -159.990, Y  +615.596, Z    +0.000, E1   -36.980, E3 -353594.991}
SPL {X  -159.990, Y  +586.905, Z    +0.000, E1   -41.264, E3 -353642.017}
SPL {X  -159.990, Y  +581.111, Z    +0.000, E1   -41.245, E3 -353656.071}
SPL {X  -159.990, Y  +576.269, Z    +0.000, E1   -41.239, E3 -353667.798}
SPL {X  -159.990, Y  +571.714, Z    +0.000, E1   -41.240, E3 -353678.826}
SPL {X  -159.990, Y  +567.050, Z    +0.000, E1   -41.238, E3 -353690.113}
SPL {X  -159.990, Y  +561.959, Z    +0.000, E1   -41.251, E3 -353702.412}
SPL {X  -159.990, Y  +555.553, Z    +0.000, E1   -41.273, E3 -353717.880}
SPL {X  -159.990, Y  +549.897, Z    +0.000, E1   -41.240, E3 -353731.610}
SPL {X  -159.990, Y  +544.775, Z    +0.000, E1   -41.260, E3 -353743.985}
SPL {X  -159.990, Y  +538.952, Z    +0.000, E1   -41.247, E3 -353758.116}
SPL {X  -159.990, Y  +534.225, Z    +0.000, E1   -41.236, E3 -353769.549}
SPL {X  -159.990, Y  +529.136, Z    +0.000, E1   -41.262, E3 -353781.825}
SPL {X  -159.990, Y  +524.776, Z    +0.000, E1   -41.225, E3 -353792.438}
SPL {X  -159.990, Y  +521.454, Z    +0.000, E1   -41.236, E3 -353800.460}
SPL {X  -159.990, Y  +515.605, Z    +0.000, E1   -41.288, E3 -353814.500}
SPL {X  -159.990, Y  +509.898, Z    +0.000, E1   -41.246, E3 -353828.361}
SPL {X  -159.990, Y  +505.215, Z    +0.000, E1   -41.261, E3 -353839.677}
SPL {X  -159.990, Y  +500.102, Z    +0.000, E1   -41.251, E3 -353852.060}
SPL {X  -159.990, Y  +495.023, Z    +0.000, E1   -41.263, E3 -353864.309}
SPL {X  -159.990, Y  +479.011, Z    +0.000, E1   -45.740, E3 -353873.691}
SPL {X  -159.990, Y  +471.379, Z    +0.000, E1   -46.435, E3 -353885.306}
SPL {X  -159.990, Y  +466.895, Z    +0.000, E1   -45.533, E3 -353899.711}
SPL {X  -159.990, Y  +462.409, Z    +0.000, E1   -44.664, E3 -353914.486}
SPL {X  -159.990, Y  +458.229, Z    +0.000, E1   -43.579, E3 -353929.968}
SPL {X  -159.990, Y  +453.434, Z    +0.000, E1   -43.227, E3 -353942.742}
SPL {X  -159.990, Y  +448.702, Z    +0.000, E1   -43.218, E3 -353953.464}
SPL {X  -159.990, Y  +444.476, Z    +0.000, E1   -43.219, E3 -353963.003}
SPL {X  -159.990, Y  +440.246, Z    +0.000, E1   -43.217, E3 -353972.560}
SPL {X  -159.990, Y  +434.411, Z    +0.000, E1   -43.246, E3 -353985.691}
SPL {X  -159.990, Y  +429.216, Z    +0.000, E1   -43.210, E3 -353997.463}
SPL {X  -159.990, Y  +424.433, Z    +0.000, E1   -43.237, E3 -354008.211}
SPL {X  -159.990, Y  +419.466, Z    +0.000, E1   -43.217, E3 -354019.451}
SPL {X  -159.990, Y  +414.585, Z    +0.000, E1   -43.233, E3 -354030.442}
SPL {X  -159.990, Y  +409.927, Z    +0.000, E1   -43.217, E3 -354040.974}
SPL {X  -159.990, Y  +405.428, Z    +0.000, E1   -43.230, E3 -354051.132}
SPL {X  -159.990, Y  +401.033, Z    +0.000, E1   -43.209, E3 -354061.087}
SPL {X  -159.990, Y  +396.968, Z    +0.000, E1   -43.221, E3 -354070.245}
SPL {X  -159.990, Y  +392.163, Z    +0.000, E1   -43.223, E3 -354081.087}
SPL {X  -159.990, Y  +387.342, Z    +0.000, E1   -43.224, E3 -354091.964}
SPL {X  -159.990, Y  +382.548, Z    +0.000, E1   -43.224, E3 -354102.787}
SPL {X  -159.922, Y  +377.835, Z    +0.000, E1   -43.211, E3 -354113.504}
SPL {X  -159.712, Y  +373.072, Z    +0.000, E1   -43.177, E3 -354124.470}
SPL {X  -159.289, Y  +367.537, Z    +0.000, E1   -43.118, E3 -354137.381}
SPL {X  -158.730, Y  +362.464, Z    +0.000, E1   -43.003, E3 -354149.413}
SPL {X  -158.182, Y  +358.518, Z    +0.000, E1   -42.902, E3 -354158.892}
SPL {X  -157.507, Y  +354.423, Z    +0.000, E1   -42.786, E3 -354168.837}
SPL {X  -156.676, Y  +350.104, Z    +0.000, E1   -42.637, E3 -354179.442}
SPL {X  -155.807, Y  +346.154, Z    +0.000, E1   -42.470, E3 -354189.270}
SPL {X  -154.777, Y  +341.993, Z    +0.000, E1   -42.302, E3 -354199.695}
SPL {X  -153.585, Y  +337.686, Z    +0.000, E1   -42.062, E3 -354210.670}
SPL {X  -152.412, Y  +333.846, Z    +0.000, E1   -41.856, E3 -354220.513}
SPL {X  -151.009, Y  +329.651, Z    +0.000, E1   -41.581, E3 -354231.412}
SPL {X  -148.356, Y  +322.607, Z    +0.000, E1   -36.121, E3 -354291.888}
ENDSPLINE

SPLINE
SPL {X  -156.487, Y  +349.204, Z    +0.000, E1   -21.338, E3 -354347.014}
SPL {X  -159.136, Y  +365.992, Z    +0.000, E1   -12.463, E3 -354357.772}
SPL {X  -159.799, Y  +374.694, Z    +0.000, E1    -7.504, E3 -354360.876}
SPL {X  -159.976, Y  +380.404, Z    +0.000, E1    -3.959, E3 -354362.409}
SPL {X  -159.990, Y  +384.773, Z    +0.000, E1    -1.003, E3 -354363.304}
SPL {X  -159.990, Y  +387.968, Z    +0.000, E1    +1.448, E3 -354363.872}
SPL {X  -159.990, Y  +391.397, Z    +0.000, E1    +4.422, E3 -354364.496}
SPL {X  -159.990, Y  +395.864, Z    +0.000, E1    +8.712, E3 -354365.584}
SPL {X  -159.990, Y  +401.273, Z    +0.000, E1   +14.176, E3 -354367.312}
SPL {X  -159.990, Y  +411.788, Z    +0.000, E1   +23.693, E3 -354372.855}
SPL {X  -159.990, Y  +438.158, Z    +0.000, E1   +37.630, E3 -354396.132}
SPL {X  -159.990, Y  +468.567, Z    +0.000, E1   +41.922, E3 -354445.476}
SPL {X  -159.990, Y  +474.616, Z    +0.000, E1   +41.909, E3 -354459.805}
SPL {X  -159.990, Y  +481.610, Z    +0.000, E1   +41.947, E3 -354476.292}
SPL {X  -159.990, Y  +488.618, Z    +0.000, E1   +41.913, E3 -354492.904}
SPL {X  -159.990, Y  +494.299, Z    +0.000, E1   +41.910, E3 -354506.339}
SPL {X  -159.990, Y  +499.538, Z    +0.000, E1   +41.904, E3 -354518.733}
SPL {X  -159.990, Y  +505.259, Z    +0.000, E1   +41.922, E3 -354532.232}
SPL {X  -159.990, Y  +511.862, Z    +0.000, E1   +41.927, E3 -354547.842}
SPL {X  -159.990, Y  +517.450, Z    +0.000, E1   +41.901, E3 -354561.090}
SPL {X  -159.990, Y  +523.027, Z    +0.000, E1   +41.926, E3 -354574.234}
SPL {X  -159.990, Y  +528.611, Z    +0.000, E1   +41.900, E3 -354587.489}
SPL {X  -159.990, Y  +533.758, Z    +0.000, E1   +41.910, E3 -354599.639}
SPL {X  -159.990, Y  +539.474, Z    +0.000, E1   +41.912, E3 -354613.166}
SPL {X  -159.990, Y  +544.879, Z    +0.000, E1   +41.899, E3 -354625.977}
SPL {X  -159.990, Y  +550.802, Z    +0.000, E1   +41.920, E3 -354639.959}
SPL {X  -159.990, Y  +556.952, Z    +0.000, E1   +41.911, E3 -354654.498}
SPL {X  -159.990, Y  +562.629, Z    +0.000, E1   +41.910, E3 -354667.916}
SPL {X  -159.990, Y  +567.682, Z    +0.000, E1   +41.901, E3 -354679.875}
SPL {X  -159.990, Y  +572.912, Z    +0.000, E1   +41.914, E3 -354692.222}
SPL {X  -159.990, Y  +578.863, Z    +0.000, E1   +41.918, E3 -354706.286}
SPL {X  -159.990, Y  +584.320, Z    +0.000, E1   +41.901, E3 -354719.233}
SPL {X  -159.990, Y  +589.217, Z    +0.000, E1   +41.901, E3 -354730.806}
SPL {X  -159.990, Y  +594.252, Z    +0.000, E1   +41.903, E3 -354742.720}
SPL {X  -159.990, Y  +598.793, Z    +0.000, E1   +41.896, E3 -354753.474}
SPL {X  -159.990, Y  +604.215, Z    +0.000, E1   +41.919, E3 -354766.254}
SPL {X  -159.990, Y  +610.545, Z    +0.000, E1   +41.917, E3 -354781.224}
SPL {X  -159.990, Y  +615.720, Z    +0.000, E1   +41.899, E3 -354793.484}
SPL {X  -159.990, Y  +620.005, Z    +0.000, E1   +41.900, E3 -354803.617}
SPL {X  -159.990, Y  +624.919, Z    +0.000, E1   +41.912, E3 -354815.225}
SPL {X  -159.990, Y  +630.816, Z    +0.000, E1   +41.915, E3 -354829.154}
SPL {X  -159.990, Y  +637.009, Z    +0.000, E1   +41.925, E3 -354843.779}
SPL {X  -159.990, Y  +642.624, Z    +0.000, E1   +41.901, E3 -354857.100}
SPL {X  -159.990, Y  +647.782, Z    +0.000, E1   +41.914, E3 -354869.268}
SPL {X  -159.990, Y  +653.094, Z    +0.000, E1   +41.905, E3 -354881.847}
SPL {X  -159.990, Y  +657.893, Z    +0.000, E1   +41.899, E3 -354893.212}
SPL {X  -159.990, Y  +662.516, Z    +0.000, E1   +41.899, E3 -354904.144}
SPL {X  -159.990, Y  +668.411, Z    +0.000, E1   +41.929, E3 -354918.037}
SPL {X  -159.968, Y  +674.139, Z    +0.000, E1   +41.898, E3 -354931.641}
SPL {X  -159.817, Y  +678.937, Z    +0.000, E1   +41.879, E3 -354943.137}
SPL {X  -159.484, Y  +684.213, Z    +0.000, E1   +41.818, E3 -354955.974}
SPL {X  -159.007, Y  +689.209, Z    +0.000, E1   +41.732, E3 -354968.278}
SPL {X  -158.327, Y  +694.511, Z    +0.000, E1   +41.622, E3 -354981.529}
SPL {X  -157.480, Y  +699.729, Z    +0.000, E1   +41.453, E3 -354994.792}
SPL {X  -156.604, Y  +704.242, Z    +0.000, E1   +41.288, E3 -355006.401}
SPL {X  -155.514, Y  +709.078, Z    +0.000, E1   +41.107, E3 -355018.955}
SPL {X  -154.232, Y  +714.035, Z    +0.000, E1   +40.861, E3 -355032.014}
SPL {X  -153.147, Y  +717.790, Z    +0.000, E1   +40.640, E3 -355042.032}
SPL {X  -151.881, Y  +721.788, Z    +0.000, E1   +40.435, E3 -355052.718}
SPL {X  -148.572, Y  +730.857, Z    +0.000, E1   +36.304, E3 -355108.927}
ENDSPLINE

SPLINE
SPL {X  -156.377, Y  +705.307, Z    +0.000, E1   +21.740, E3 -355163.176}
SPL {X  -159.301, Y  +686.331, Z    +0.000, E1   +11.648, E3 -355175.820}
SPL {X  -159.936, Y  +675.651, Z    +0.000, E1    +5.377, E3 -355179.536}
SPL {X  -159.990, Y  +670.142, Z    +0.000, E1    +1.740, E3 -355180.836}
SPL {X  -159.990, Y  +666.629, Z    +0.000, E1    -0.827, E3 -355181.485}
SPL {X  -159.990, Y  +662.407, Z    +0.000, E1    -4.406, E3 -355182.336}
SPL {X  -159.990, Y  +657.382, Z    +0.000, E1    -9.217, E3 -355183.718}
SPL {X  -159.990, Y  +653.255, Z    +0.000, E1   -13.347, E3 -355185.047}
SPL {X  -159.990, Y  +646.242, Z    +0.000, E1   -19.956, E3 -355188.120}
SPL {X  -159.990, Y  +624.365, Z    +0.000, E1   -33.860, E3 -355206.022}
SPL {X  -159.990, Y  +615.596, Z    +0.000, E1   -36.980, E3 -355215.680}
SPL {X  -159.990, Y  +586.905, Z    +0.000, E1   -41.264, E3 -355262.707}
SPL {X  -159.990, Y  +581.111, Z    +0.000, E1   -41.245, E3 -355276.761}
SPL {X  -159.990, Y  +576.269, Z    +0.000, E1   -41.239, E3 -355288.488}
SPL {X  -159.990, Y  +571.714, Z    +0.000, E1   -41.240, E3 -355299.516}
SPL {X  -159.990, Y  +567.050, Z    +0.000, E1   -41.238, E3 -355310.803}
SPL {X  -159.990, Y  +561.959, Z    +0.000, E1   -41.251, E3 -355323.101}
SPL {X  -159.990, Y  +555.553, Z    +0.000, E1   -41.273, E3 -355338.570}
SPL {X  -159.990, Y  +549.897, Z    +0.000, E1   -41.240, E3 -355352.300}
SPL {X  -159.990, Y  +544.775, Z    +0.000, E1   -41.260, E3 -355364.675}
SPL {X  -159.990, Y  +540.176, Z    +0.000, E1   -41.224, E3 -355375.883}
SPL {X  -159.990, Y  +534.009, Z    +0.000, E1   -41.300, E3 -355390.669}
SPL {X  -159.990, Y  +526.579, Z    +0.000, E1   -41.262, E3 -355408.706}
SPL {X  -159.990, Y  +521.454, Z    +0.000, E1   -41.236, E3 -355421.150}
SPL {X  -159.990, Y  +515.605, Z    +0.000, E1   -41.288, E3 -355435.189}
SPL {X  -159.990, Y  +509.898, Z    +0.000, E1   -41.246, E3 -355449.050}
SPL {X  -159.990, Y  +505.215, Z    +0.000, E1   -41.261, E3 -355460.366}
SPL {X  -159.990, Y  +500.102, Z    +0.000, E1   -41.251, E3 -355472.750}
SPL {X  -159.990, Y  +495.023, Z    +0.000, E1   -41.263, E3 -355484.998}
SPL {X  -159.990, Y  +479.011, Z    +0.000, E1   -45.740, E3 -355494.380}
SPL {X  -159.990, Y  +471.379, Z    +0.000, E1   -46.435, E3 -355505.996}
SPL {X  -159.990, Y  +465.881, Z    +0.000, E1   -45.385, E3 -355523.599}
SPL {X  -159.990, Y  +461.571, Z    +0.000, E1   -44.440, E3 -355538.124}
SPL {X  -159.990, Y  +458.229, Z    +0.000, E1   -43.579, E3 -355550.658}
SPL {X  -159.990, Y  +453.434, Z    +0.000, E1   -43.227, E3 -355563.432}
SPL {X  -159.990, Y  +448.702, Z    +0.000, E1   -43.218, E3 -355574.154}
SPL {X  -159.990, Y  +442.224, Z    +0.000, E1   -43.270, E3 -355588.704}
SPL {X  -159.990, Y  +435.724, Z    +0.000, E1   -43.218, E3 -355603.462}
SPL {X  -159.990, Y  +430.527, Z    +0.000, E1   -43.236, E3 -355615.151}
SPL {X  -159.990, Y  +424.433, Z    +0.000, E1   -43.237, E3 -355628.901}
SPL {X  -159.990, Y  +419.466, Z    +0.000, E1   -43.217, E3 -355640.140}
SPL {X  -159.990, Y  +414.585, Z    +0.000, E1   -43.233, E3 -355651.132}
SPL {X  -159.990, Y  +409.927, Z    +0.000, E1   -43.217, E3 -355661.664}
SPL {X  -159.990, Y  +405.428, Z    +0.000, E1   -43.230, E3 -355671.822}
SPL {X  -159.990, Y  +401.033, Z    +0.000, E1   -43.209, E3 -355681.776}
SPL {X  -159.990, Y  +396.968, Z    +0.000, E1   -43.221, E3 -355690.934}
SPL {X  -159.990, Y  +392.163, Z    +0.000, E1   -43.223, E3 -355701.776}
SPL {X  -159.990, Y  +387.342, Z    +0.000, E1   -43.224, E3 -355712.654}
SPL {X  -159.990, Y  +382.548, Z    +0.000, E1   -43.224, E3 -355723.477}
SPL {X  -159.922, Y  +377.835, Z    +0.000, E1   -43.211, E3 -355734.193}
SPL {X  -159.608, Y  +371.448, Z    +0.000, E1   -43.200, E3 -355748.870}
SPL {X  -158.905, Y  +363.898, Z    +0.000, E1   -43.073, E3 -355766.638}
SPL {X  -158.182, Y  +358.518, Z    +0.000, E1   -42.902, E3 -355779.581}
SPL {X  -157.507, Y  +354.423, Z    +0.000, E1   -42.786, E3 -355789.527}
SPL {X  -156.676, Y  +350.104, Z    +0.000, E1   -42.637, E3 -355800.132}
SPL {X  -155.807, Y  +346.154, Z    +0.000, E1   -42.470, E3 -355809.959}
SPL {X  -154.777, Y  +341.993, Z    +0.000, E1   -42.302, E3 -355820.384}
SPL {X  -153.585, Y  +337.686, Z    +0.000, E1   -42.062, E3 -355831.360}
SPL {X  -152.412, Y  +333.846, Z    +0.000, E1   -41.856, E3 -355841.202}
SPL {X  -151.009, Y  +329.651, Z    +0.000, E1   -41.581, E3 -355852.102}
SPL {X  -148.356, Y  +322.607, Z    +0.000, E1   -36.121, E3 -355912.578}
ENDSPLINE

SPLINE
SPL {X  -156.487, Y  +349.204, Z    +0.000, E1   -21.338, E3 -355967.704}
SPL {X  -159.136, Y  +365.992, Z    +0.000, E1   -12.463, E3 -355978.462}
SPL {X  -159.799, Y  +374.694, Z    +0.000, E1    -7.504, E3 -355981.566}
SPL {X  -159.976, Y  +380.404, Z    +0.000, E1    -3.959, E3 -355983.099}
SPL {X  -159.990, Y  +384.773, Z    +0.000, E1    -1.003, E3 -355983.993}
SPL {X  -159.990, Y  +387.968, Z    +0.000, E1    +1.448, E3 -355984.562}
SPL {X  -159.990, Y  +391.397, Z    +0.000, E1    +4.422, E3 -355985.186}
SPL {X  -159.990, Y  +395.864, Z    +0.000, E1    +8.712, E3 -355986.274}
SPL {X  -159.990, Y  +401.273, Z    +0.000, E1   +14.176, E3 -355988.001}
SPL {X  -159.990, Y  +411.788, Z    +0.000, E1   +23.693, E3 -355993.544}
SPL {X  -159.990, Y  +438.158, Z    +0.000, E1   +37.630, E3 -356016.822}
SPL {X  -159.990, Y  +469.969, Z    +0.000, E1   +41.961, E3 -356069.423}
SPL {X  -159.990, Y  +477.498, Z    +0.000, E1   +41.916, E3 -356087.306}
SPL {X  -159.990, Y  +483.140, Z    +0.000, E1   +41.902, E3 -356100.662}
SPL {X  -159.990, Y  +488.618, Z    +0.000, E1   +41.913, E3 -356113.594}
SPL {X  -159.990, Y  +494.299, Z    +0.000, E1   +41.910, E3 -356127.028}
SPL {X  -159.990, Y  +499.538, Z    +0.000, E1   +41.904, E3 -356139.422}
SPL {X  -159.990, Y  +505.259, Z    +0.000, E1   +41.922, E3 -356152.922}
SPL {X  -159.990, Y  +511.862, Z    +0.000, E1   +41.927, E3 -356168.532}
SPL {X  -159.990, Y  +517.450, Z    +0.000, E1   +41.901, E3 -356181.780}
SPL {X  -159.990, Y  +523.027, Z    +0.000, E1   +41.926, E3 -356194.924}
SPL {X  -159.990, Y  +528.611, Z    +0.000, E1   +41.900, E3 -356208.179}
SPL {X  -159.990, Y  +533.758, Z    +0.000, E1   +41.910, E3 -356220.328}
SPL {X  -159.990, Y  +539.474, Z    +0.000, E1   +41.912, E3 -356233.856}
SPL {X  -159.990, Y  +544.879, Z    +0.000, E1   +41.899, E3 -356246.667}
SPL {X  -159.990, Y  +550.802, Z    +0.000, E1   +41.920, E3 -356260.648}
SPL {X  -159.990, Y  +556.952, Z    +0.000, E1   +41.911, E3 -356275.188}
SPL {X  -159.990, Y  +562.629, Z    +0.000, E1   +41.910, E3 -356288.606}
SPL {X  -159.990, Y  +567.682, Z    +0.000, E1   +41.901, E3 -356300.565}
SPL {X  -159.990, Y  +572.912, Z    +0.000, E1   +41.914, E3 -356312.912}
SPL {X  -159.990, Y  +578.863, Z    +0.000, E1   +41.918, E3 -356326.976}
SPL {X  -159.990, Y  +584.320, Z    +0.000, E1   +41.901, E3 -356339.923}
SPL {X  -159.990, Y  +589.217, Z    +0.000, E1   +41.901, E3 -356351.495}
SPL {X  -159.990, Y  +594.252, Z    +0.000, E1   +41.903, E3 -356363.410}
SPL {X  -159.990, Y  +598.793, Z    +0.000, E1   +41.896, E3 -356374.164}
SPL {X  -159.990, Y  +604.215, Z    +0.000, E1   +41.919, E3 -356386.944}
SPL {X  -159.990, Y  +610.545, Z    +0.000, E1   +41.917, E3 -356401.914}
SPL {X  -159.990, Y  +615.720, Z    +0.000, E1   +41.899, E3 -356414.174}
SPL {X  -159.990, Y  +621.417, Z    +0.000, E1   +41.931, E3 -356427.611}
SPL {X  -159.990, Y  +627.900, Z    +0.000, E1   +41.914, E3 -356442.950}
SPL {X  -159.990, Y  +632.270, Z    +0.000, E1   +41.887, E3 -356453.326}
SPL {X  -159.990, Y  +637.009, Z    +0.000, E1   +41.925, E3 -356464.469}
SPL {X  -159.990, Y  +642.624, Z    +0.000, E1   +41.901, E3 -356477.790}
SPL {X  -159.990, Y  +647.782, Z    +0.000, E1   +41.914, E3 -356489.958}
SPL {X  -159.990, Y  +653.094, Z    +0.000, E1   +41.905, E3 -356502.536}
SPL {X  -159.990, Y  +657.893, Z    +0.000, E1   +41.899, E3 -356513.902}
SPL {X  -159.990, Y  +662.516, Z    +0.000, E1   +41.899, E3 -356524.833}
SPL {X  -159.990, Y  +666.974, Z    +0.000, E1   +41.897, E3 -356535.378}
SPL {X  -159.984, Y  +672.859, Z    +0.000, E1   +41.934, E3 -356549.239}
SPL {X  -159.817, Y  +678.937, Z    +0.000, E1   +41.879, E3 -356563.827}
SPL {X  -159.484, Y  +684.213, Z    +0.000, E1   +41.818, E3 -356576.663}
SPL {X  -159.007, Y  +689.209, Z    +0.000, E1   +41.732, E3 -356588.968}
SPL {X  -158.485, Y  +693.390, Z    +0.000, E1   +41.627, E3 -356599.421}
SPL {X  -157.663, Y  +698.690, Z    +0.000, E1   +41.523, E3 -356612.783}
SPL {X  -156.604, Y  +704.242, Z    +0.000, E1   +41.288, E3 -356627.091}
SPL {X  -155.831, Y  +707.744, Z    +0.000, E1   +41.132, E3 -356636.211}
SPL {X  -155.167, Y  +710.488, Z    +0.000, E1   +41.008, E3 -356643.389}
SPL {X  -154.232, Y  +714.035, Z    +0.000, E1   +40.861, E3 -356652.703}
SPL {X  -153.147, Y  +717.790, Z    +0.000, E1   +40.640, E3 -356662.722}
SPL {X  -151.881, Y  +721.788, Z    +0.000, E1   +40.435, E3 -356673.408}
SPL {X  -148.572, Y  +730.857, Z    +0.000, E1   +36.304, E3 -356729.617}
ENDSPLINE

SPLINE
SPL {X  -154.420, Y  +713.347, Z    +0.000, E1   +25.698, E3 -356775.041}
SPL {X  -156.970, Y  +702.437, Z    +0.000, E1   +20.224, E3 -356786.737}
SPL {X  -159.301, Y  +686.331, Z    +0.000, E1   +11.648, E3 -356796.510}
SPL {X  -159.936, Y  +675.651, Z    +0.000, E1    +5.377, E3 -356800.226}
SPL {X  -159.990, Y  +670.142, Z    +0.000, E1    +1.740, E3 -356801.525}
SPL {X  -159.990, Y  +666.629, Z    +0.000, E1    -0.827, E3 -356802.175}
SPL {X  -159.990, Y  +662.407, Z    +0.000, E1    -4.406, E3 -356803.025}
SPL {X  -159.990, Y  +655.884, Z    +0.000, E1   -10.601, E3 -356804.891}
SPL {X  -159.990, Y  +643.833, Z    +0.000, E1   -21.883, E3 -356810.520}
SPL {X  -159.990, Y  +617.235, Z    +0.000, E1   -36.481, E3 -356834.420}
SPL {X  -159.990, Y  +586.905, Z    +0.000, E1   -41.264, E3 -356883.396}
SPL {X  -159.990, Y  +581.111, Z    +0.000, E1   -41.245, E3 -356897.450}
SPL {X  -159.990, Y  +576.269, Z    +0.000, E1   -41.239, E3 -356909.178}
SPL {X  -159.990, Y  +571.714, Z    +0.000, E1   -41.240, E3 -356920.206}
SPL {X  -159.990, Y  +567.050, Z    +0.000, E1   -41.238, E3 -356931.493}
SPL {X  -159.990, Y  +561.959, Z    +0.000, E1   -41.251, E3 -356943.791}
SPL {X  -159.990, Y  +555.553, Z    +0.000, E1   -41.273, E3 -356959.259}
SPL {X  -159.990, Y  +549.897, Z    +0.000, E1   -41.240, E3 -356972.990}
SPL {X  -159.990, Y  +544.775, Z    +0.000, E1   -41.260, E3 -356985.364}
SPL {X  -159.990, Y  +540.176, Z    +0.000, E1   -41.224, E3 -356996.573}
SPL {X  -159.990, Y  +535.325, Z    +0.000, E1   -41.260, E3 -357008.237}
SPL {X  -159.990, Y  +529.136, Z    +0.000, E1   -41.262, E3 -357023.204}
SPL {X  -159.990, Y  +522.690, Z    +0.000, E1   -41.265, E3 -357038.804}
SPL {X  -159.990, Y  +516.698, Z    +0.000, E1   -41.259, E3 -357053.278}
SPL {X  -159.990, Y  +510.896, Z    +0.000, E1   -41.267, E3 -357067.296}
SPL {X  -159.990, Y  +505.215, Z    +0.000, E1   -41.261, E3 -357081.056}
SPL {X  -159.990, Y  +500.102, Z    +0.000, E1   -41.251, E3 -357093.439}
SPL {X  -159.990, Y  +495.023, Z    +0.000, E1   -41.263, E3 -357105.688}
SPL {X  -159.990, Y  +479.011, Z    +0.000, E1   -45.740, E3 -357115.070}
SPL {X  -159.990, Y  +471.379, Z    +0.000, E1   -46.435, E3 -357126.685}
SPL {X  -159.990, Y  +466.895, Z    +0.000, E1   -45.533, E3 -357141.090}
SPL {X  -159.990, Y  +462.409, Z    +0.000, E1   -44.664, E3 -357155.865}
SPL {X  -159.990, Y  +458.229, Z    +0.000, E1   -43.579, E3 -357171.347}
SPL {X  -159.990, Y  +453.434, Z    +0.000, E1   -43.227, E3 -357184.122}
SPL {X  -159.990, Y  +448.702, Z    +0.000, E1   -43.218, E3 -357194.844}
SPL {X  -159.990, Y  +442.224, Z    +0.000, E1   -43.270, E3 -357209.394}
SPL {X  -159.990, Y  +435.724, Z    +0.000, E1   -43.218, E3 -357224.152}
SPL {X  -159.990, Y  +430.527, Z    +0.000, E1   -43.236, E3 -357235.841}
SPL {X  -159.990, Y  +424.433, Z    +0.000, E1   -43.237, E3 -357249.590}
SPL {X  -159.990, Y  +419.466, Z    +0.000, E1   -43.217, E3 -357260.830}
SPL {X  -159.990, Y  +414.585, Z    +0.000, E1   -43.233, E3 -357271.822}
SPL {X  -159.990, Y  +409.927, Z    +0.000, E1   -43.217, E3 -357282.353}
SPL {X  -159.990, Y  +405.428, Z    +0.000, E1   -43.230, E3 -357292.512}
SPL {X  -159.990, Y  +398.518, Z    +0.000, E1   -43.261, E3 -357308.066}
SPL {X  -159.990, Y  +392.163, Z    +0.000, E1   -43.223, E3 -357322.466}
SPL {X  -159.990, Y  +387.342, Z    +0.000, E1   -43.224, E3 -357333.343}
SPL {X  -159.990, Y  +382.548, Z    +0.000, E1   -43.224, E3 -357344.166}
SPL {X  -159.922, Y  +377.835, Z    +0.000, E1   -43.211, E3 -357354.883}
SPL {X  -159.712, Y  +373.072, Z    +0.000, E1   -43.177, E3 -357365.849}
SPL {X  -159.289, Y  +367.537, Z    +0.000, E1   -43.118, E3 -357378.761}
SPL {X  -158.730, Y  +362.464, Z    +0.000, E1   -43.003, E3 -357390.793}
SPL {X  -158.182, Y  +358.518, Z    +0.000, E1   -42.902, E3 -357400.271}
SPL {X  -157.507, Y  +354.423, Z    +0.000, E1   -42.786, E3 -357410.216}
SPL {X  -156.676, Y  +350.104, Z    +0.000, E1   -42.637, E3 -357420.822}
SPL {X  -155.489, Y  +344.819, Z    +0.000, E1   -42.446, E3 -357433.945}
SPL {X  -153.911, Y  +338.816, Z    +0.000, E1   -42.155, E3 -357449.121}
SPL {X  -152.412, Y  +333.846, Z    +0.000, E1   -41.856, E3 -357461.892}
SPL {X  -151.009, Y  +329.651, Z    +0.000, E1   -41.581, E3 -357472.792}
SPL {X  -148.356, Y  +322.607, Z    +0.000, E1   -36.121, E3 -357533.267}
ENDSPLINE

SPLINE
SPL {X  -156.487, Y  +349.204, Z    +0.000, E1   -21.338, E3 -357588.393}
SPL {X  -159.136, Y  +365.992, Z    +0.000, E1   -12.463, E3 -357599.152}
SPL {X  -159.799, Y  +374.694, Z    +0.000, E1    -7.504, E3 -357602.255}
SPL {X  -159.976, Y  +380.404, Z    +0.000, E1    -3.959, E3 -357603.788}
SPL {X  -159.990, Y  +384.773, Z    +0.000, E1    -1.003, E3 -357604.683}
SPL {X  -159.990, Y  +387.968, Z    +0.000, E1    +1.448, E3 -357605.251}
SPL {X  -159.990, Y  +391.397, Z    +0.000, E1    +4.422, E3 -357605.875}
SPL {X  -159.990, Y  +395.864, Z    +0.000, E1    +8.712, E3 -357606.964}
SPL {X  -159.990, Y  +401.273, Z    +0.000, E1   +14.176, E3 -357608.691}
SPL {X  -159.990, Y  +409.369, Z    +0.000, E1   +21.807, E3 -357612.483}
SPL {X  -159.990, Y  +436.107, Z    +0.000, E1   +36.921, E3 -357635.408}
SPL {X  -159.990, Y  +465.724, Z    +0.000, E1   +41.883, E3 -357680.206}
SPL {X  -159.990, Y  +470.837, Z    +0.000, E1   +41.927, E3 -357692.221}
SPL {X  -159.990, Y  +477.498, Z    +0.000, E1   +41.916, E3 -357707.996}
SPL {X  -159.990, Y  +483.140, Z    +0.000, E1   +41.902, E3 -357721.352}
SPL {X  -159.990, Y  +488.618, Z    +0.000, E1   +41.913, E3 -357734.284}
SPL {X  -159.990, Y  +494.299, Z    +0.000, E1   +41.910, E3 -357747.718}
SPL {X  -159.990, Y  +499.538, Z    +0.000, E1   +41.904, E3 -357760.112}
SPL {X  -159.990, Y  +505.259, Z    +0.000, E1   +41.922, E3 -357773.611}
SPL {X  -159.990, Y  +511.862, Z    +0.000, E1   +41.927, E3 -357789.222}
SPL {X  -159.990, Y  +517.450, Z    +0.000, E1   +41.901, E3 -357802.469}
SPL {X  -159.990, Y  +523.027, Z    +0.000, E1   +41.926, E3 -357815.613}
SPL {X  -159.990, Y  +528.611, Z    +0.000, E1   +41.900, E3 -357828.869}
SPL {X  -159.990, Y  +533.758, Z    +0.000, E1   +41.910, E3 -357841.018}
SPL {X  -159.990, Y  +539.474, Z    +0.000, E1   +41.912, E3 -357854.545}
SPL {X  -159.990, Y  +544.879, Z    +0.000, E1   +41.899, E3 -357867.357}
SPL {X  -159.990, Y  +550.802, Z    +0.000, E1   +41.920, E3 -357881.338}
SPL {X  -159.990, Y  +556.952, Z    +0.000, E1   +41.911, E3 -357895.877}
SPL {X  -159.990, Y  +562.629, Z    +0.000, E1   +41.910, E3 -357909.295}
SPL {X  -159.990, Y  +567.682, Z    +0.000, E1   +41.901, E3 -357921.254}
SPL {X  -159.990, Y  +572.912, Z    +0.000, E1   +41.914, E3 -357933.601}
SPL {X  -159.990, Y  +578.863, Z    +0.000, E1   +41.918, E3 -357947.666}
SPL {X  -159.990, Y  +584.320, Z    +0.000, E1   +41.901, E3 -357960.612}
SPL {X  -159.990, Y  +589.217, Z    +0.000, E1   +41.901, E3 -357972.185}
SPL {X  -159.990, Y  +594.252, Z    +0.000, E1   +41.903, E3 -357984.100}
SPL {X  -159.990, Y  +598.793, Z    +0.000, E1   +41.896, E3 -357994.854}
SPL {X  -159.990, Y  +604.215, Z    +0.000, E1   +41.919, E3 -358007.634}
SPL {X  -159.990, Y  +609.216, Z    +0.000, E1   +41.890, E3 -358019.502}
SPL {X  -159.990, Y  +614.570, Z    +0.000, E1   +41.926, E3 -358032.107}
SPL {X  -159.990, Y  +620.005, Z    +0.000, E1   +41.900, E3 -358044.997}
SPL {X  -159.990, Y  +624.919, Z    +0.000, E1   +41.912, E3 -358056.604}
SPL {X  -159.990, Y  +629.282, Z    +0.000, E1   +41.888, E3 -358066.945}
SPL {X  -159.990, Y  +632.270, Z    +0.000, E1   +41.887, E3 -358074.016}
SPL {X  -159.990, Y  +637.009, Z    +0.000, E1   +41.925, E3 -358085.159}
SPL {X  -159.990, Y  +642.624, Z    +0.000, E1   +41.901, E3 -358098.479}
SPL {X  -159.990, Y  +647.782, Z    +0.000, E1   +41.914, E3 -358110.648}
SPL {X  -159.990, Y  +653.094, Z    +0.000, E1   +41.905, E3 -358123.226}
SPL {X  -159.990, Y  +657.893, Z    +0.000, E1   +41.899, E3 -358134.592}
SPL {X  -159.990, Y  +662.516, Z    +0.000, E1   +41.899, E3 -358145.523}
SPL {X  -159.990, Y  +668.411, Z    +0.000, E1   +41.929, E3 -358159.417}
SPL {X  -159.968, Y  +674.139, Z    +0.000, E1   +41.898, E3 -358173.021}
SPL {X  -159.817, Y  +678.937, Z    +0.000, E1   +41.879, E3 -358184.517}
SPL {X  -159.484, Y  +684.213, Z    +0.000, E1   +41.818, E3 -358197.353}
SPL {X  -159.007, Y  +689.209, Z    +0.000, E1   +41.732, E3 -358209.658}
SPL {X  -158.327, Y  +694.511, Z    +0.000, E1   +41.622, E3 -358222.909}
SPL {X  -157.480, Y  +699.729, Z    +0.000, E1   +41.453, E3 -358236.172}
SPL {X  -156.604, Y  +704.242, Z    +0.000, E1   +41.288, E3 -358247.780}
SPL {X  -155.831, Y  +707.744, Z    +0.000, E1   +41.132, E3 -358256.900}
SPL {X  -155.167, Y  +710.488, Z    +0.000, E1   +41.008, E3 -358264.078}
SPL {X  -154.232, Y  +714.035, Z    +0.000, E1   +40.861, E3 -358273.393}
SPL {X  -153.147, Y  +717.790, Z    +0.000, E1   +40.640, E3 -358283.411}
SPL {X  -151.881, Y  +721.788, Z    +0.000, E1   +40.435, E3 -358294.098}
SPL {X  -148.572, Y  +730.857, Z    +0.000, E1   +36.304, E3 -358350.307}
ENDSPLINE

SPLINE
SPL {X  -156.377, Y  +705.307, Z    +0.000, E1   +21.740, E3 -358404.555}
SPL {X  -158.965, Y  +689.585, Z    +0.000, E1   +13.405, E3 -358415.713}
SPL {X  -159.884, Y  +677.314, Z    +0.000, E1    +6.475, E3 -358420.426}
SPL {X  -159.990, Y  +670.142, Z    +0.000, E1    +1.740, E3 -358422.215}
SPL {X  -159.990, Y  +666.629, Z    +0.000, E1    -0.827, E3 -358422.864}
SPL {X  -159.990, Y  +662.407, Z    +0.000, E1    -4.406, E3 -358423.715}
SPL {X  -159.990, Y  +657.382, Z    +0.000, E1    -9.217, E3 -358425.097}
SPL {X  -159.990, Y  +653.255, Z    +0.000, E1   -13.347, E3 -358426.426}
SPL {X  -159.990, Y  +646.242, Z    +0.000, E1   -19.956, E3 -358429.500}
SPL {X  -159.990, Y  +624.365, Z    +0.000, E1   -33.860, E3 -358447.401}
SPL {X  -159.990, Y  +615.596, Z    +0.000, E1   -36.980, E3 -358457.060}
SPL {X  -159.990, Y  +588.349, Z    +0.000, E1   -41.235, E3 -358500.638}
SPL {X  -159.990, Y  +582.302, Z    +0.000, E1   -41.281, E3 -358515.205}
SPL {X  -159.990, Y  +576.269, Z    +0.000, E1   -41.239, E3 -358529.867}
SPL {X  -159.990, Y  +571.714, Z    +0.000, E1   -41.240, E3 -358540.895}
SPL {X  -159.990, Y  +567.050, Z    +0.000, E1   -41.238, E3 -358552.182}
SPL {X  -159.990, Y  +561.959, Z    +0.000, E1   -41.251, E3 -358564.481}
SPL {X  -159.990, Y  +555.553, Z    +0.000, E1   -41.273, E3 -358579.949}
SPL {X  -159.990, Y  +549.897, Z    +0.000, E1   -41.240, E3 -358593.679}
SPL {X  -159.990, Y  +544.775, Z    +0.000, E1   -41.260, E3 -358606.054}
SPL {X  -159.990, Y  +538.952, Z    +0.000, E1   -41.247, E3 -358620.185}
SPL {X  -159.990, Y  +532.945, Z    +0.000, E1   -41.264, E3 -358634.673}
SPL {X  -159.990, Y  +526.579, Z    +0.000, E1   -41.262, E3 -358650.085}
SPL {X  -159.990, Y  +521.454, Z    +0.000, E1   -41.236, E3 -358662.529}
SPL {X  -159.990, Y  +516.698, Z    +0.000, E1   -41.259, E3 -358673.968}
SPL {X  -159.990, Y  +510.896, Z    +0.000, E1   -41.267, E3 -358687.986}
SPL {X  -159.990, Y  +505.215, Z    +0.000, E1   -41.261, E3 -358701.746}
SPL {X  -159.990, Y  +498.837, Z    +0.000, E1   -41.283, E3 -358717.134}
SPL {X  -159.990, Y  +493.848, Z    +0.000, E1   -41.241, E3 -358729.254}
SPL {X  -159.990, Y  +474.734, Z    +0.000, E1   -46.319, E3 -358741.178}
SPL {X  -159.990, Y  +469.870, Z    +0.000, E1   -46.059, E3 -358752.400}
SPL {X  -159.990, Y  +465.881, Z    +0.000, E1   -45.385, E3 -358764.978}
SPL {X  -159.990, Y  +461.571, Z    +0.000, E1   -44.440, E3 -358779.503}
SPL {X  -159.990, Y  +458.229, Z    +0.000, E1   -43.579, E3 -358792.037}
SPL {X  -159.990, Y  +453.434, Z    +0.000, E1   -43.227, E3 -358804.811}
SPL {X  -159.990, Y  +448.702, Z    +0.000, E1   -43.218, E3 -358815.533}
SPL {X  -159.990, Y  +442.224, Z    +0.000, E1   -43.270, E3 -358830.083}
SPL {X  -159.990, Y  +435.724, Z    +0.000, E1   -43.218, E3 -358844.841}
SPL {X  -159.990, Y  +430.527, Z    +0.000, E1   -43.236, E3 -358856.531}
SPL {X  -159.990, Y  +424.433, Z    +0.000, E1   -43.237, E3 -358870.280}
SPL {X  -159.990, Y  +419.466, Z    +0.000, E1   -43.217, E3 -358881.519}
SPL {X  -159.990, Y  +414.585, Z    +0.000, E1   -43.233, E3 -358892.511}
SPL {X  -159.990, Y  +409.927, Z    +0.000, E1   -43.217, E3 -358903.043}
SPL {X  -159.990, Y  +405.428, Z    +0.000, E1   -43.230, E3 -358913.201}
SPL {X  -159.990, Y  +398.518, Z    +0.000, E1   -43.261, E3 -358928.756}
SPL {X  -159.990, Y  +392.163, Z    +0.000, E1   -43.223, E3 -358943.156}
SPL {X  -159.990, Y  +387.342, Z    +0.000, E1   -43.224, E3 -358954.033}
SPL {X  -159.990, Y  +382.548, Z    +0.000, E1   -43.224, E3 -358964.856}
SPL {X  -159.922, Y  +377.835, Z    +0.000, E1   -43.211, E3 -358975.573}
SPL {X  -159.712, Y  +373.072, Z    +0.000, E1   -43.177, E3 -358986.539}
SPL {X  -159.289, Y  +367.537, Z    +0.000, E1   -43.118, E3 -358999.450}
SPL {X  -158.730, Y  +362.464, Z    +0.000, E1   -43.003, E3 -359011.482}
SPL {X  -158.182, Y  +358.518, Z    +0.000, E1   -42.902, E3 -359020.961}
SPL {X  -157.507, Y  +354.423, Z    +0.000, E1   -42.786, E3 -359030.906}
SPL {X  -156.676, Y  +350.104, Z    +0.000, E1   -42.637, E3 -359041.511}
SPL {X  -155.807, Y  +346.154, Z    +0.000, E1   -42.470, E3 -359051.339}
SPL {X  -154.777, Y  +341.993, Z    +0.000, E1   -42.302, E3 -359061.764}
SPL {X  -153.585, Y  +337.686, Z    +0.000, E1   -42.062, E3 -359072.739}
SPL {X  -152.412, Y  +333.846, Z    +0.000, E1   -41.856, E3 -359082.582}
SPL {X  -151.009, Y  +329.651, Z    +0.000, E1   -41.581, E3 -359093.481}
SPL {X  -148.356, Y  +322.607, Z    +0.000, E1   -36.121, E3 -359153.957}
ENDSPLINE

